NETWORK
TITLE = Hys Calculation
//Level Hys Absolute
      L     #Param.L_Hi_Lim;
      L     #Param.L_Lo_Lim;
      -R;
      L     100.0;
      /R;
      L     #Param.L_Hys;
      *R;
      T     #L_Hys_Abs;
//Tank High Level
      L     #Param.SP_Level_HL;
      L     #L_Hys_Abs;
      -R;
      T     #Hys_Level_HL;
//Tank Mid Level
      L     #Param.SP_Level_ML;
      L     #L_Hys_Abs;
      -R;
      T     #Hys_Level_ML;
//Tank Low Level
      L     #Param.SP_Level_LL;
      L     #L_Hys_Abs;
      +R;
      T     #Hys_Level_LL;


REGION Network 3: Level Tank
   RUNG wire#powerrail
      Contact( #alwaysON )
      wire#w1
      { S7_Templates := "SrcType := Real" } LE_Contact(in1 := #Param.SP_Level_HL, in2 := #IN_LT01)
      S_Coil( #State.Tank_HL )
   END_RUNG
   RUNG wire#w1
      { S7_Templates := "SrcType := Real" } GT_Contact(in1 := #Hys_Level_HL, in2 := #IN_LT01)
      R_Coil( #State.Tank_HL )
   END_RUNG
   RUNG wire#w1
      { S7_Templates := "SrcType := Real" } LE_Contact(in1 := #Param.SP_Level_ML, in2 := #IN_LT01)
      S_Coil( #State.Tank_ML )
   END_RUNG
   RUNG wire#w1
      { S7_Templates := "SrcType := Real" } GT_Contact(in1 := #Hys_Level_ML, in2 := #IN_LT01)
      R_Coil( #State.Tank_ML )
   END_RUNG
   RUNG wire#w1
      { S7_Templates := "SrcType := Real" } GE_Contact(in1 := #Param.SP_Level_LL, in2 := #IN_LT01)
      S_Coil( #State.Tank_LL )
   END_RUNG
   RUNG wire#w1
      { S7_Templates := "SrcType := Real" } LT_Contact(in1 := #Hys_Level_LL, in2 := #IN_LT01)
      R_Coil( #State.Tank_LL )
   END_RUNG
   // the same network as SCL:
   IF #alwaysON AND (#Param.SP_Level_HL <= #IN_LT01) THEN #State.Tank_HL := TRUE; END_IF;
   IF #alwaysON AND (#Hys_Level_HL > #IN_LT01) THEN #State.Tank_HL := FALSE; END_IF;
   IF #alwaysON AND (#Param.SP_Level_ML <= #IN_LT01) THEN #State.Tank_ML := TRUE; END_IF;
   IF #alwaysON AND (#Hys_Level_ML > #IN_LT01) THEN #State.Tank_ML := FALSE; END_IF;
   IF #alwaysON AND (#Param.SP_Level_LL >= #IN_LT01) THEN #State.Tank_LL := TRUE; END_IF;
   IF #alwaysON AND (#Hys_Level_LL < #IN_LT01) THEN #State.Tank_LL := FALSE; END_IF;
END_REGION

REGION Network 4: Reset Command Inload
   RUNG wire#powerrail
      Contact( #alwaysON )
      Contact( #State.Tank_HL )
      P_Trig( #r.PosE1 )
      wire#w1
      R_Coil( #Cmd.Inload )
   END_RUNG
   RUNG wire#w1
      R_Coil( #Actuator.LCS_OnOff )
   END_RUNG
   // the same network as SCL:
   #_w1 := #alwaysON AND #State.Tank_HL;
   #_w2 := #_w1 AND NOT #r.PosE1;   // rising edge
   #r.PosE1 := #_w1;
   IF #_w2 THEN
       #Cmd.Inload := FALSE;
       #Actuator.LCS_OnOff := FALSE;
   END_IF;
END_REGION

REGION Network 5: Inload from LCS ON-OFF
   RUNG wire#powerrail
      Contact( #alwaysON )
      wire#w1
      Contact( #"LCS Start" )
      S_Coil( #Actuator.LCS_OnOff )
   END_RUNG
   RUNG wire#w1
      Contact( #"LCS Stop" )
      R_Coil( #Actuator.LCS_OnOff )
   END_RUNG
   // the same network as SCL:
   IF #alwaysON AND #"LCS Start" THEN #Actuator.LCS_OnOff := TRUE; END_IF;
   IF #alwaysON AND #"LCS Stop" THEN #Actuator.LCS_OnOff := FALSE; END_IF;
END_REGION

REGION Network 6: Command Inload Material to Buffer Tank
   RUNG wire#powerrail
      Contact( #alwaysON )
      wire#w1
      I_Contact( #State.Tank_HL )
      I_Contact( #"Inload Busy" )
      I_Contact( #State.Tank_inCIP )
      I_Contact( #State.Line_inCIP )
      Coil( #State.Inload_Enable )
   END_RUNG
   RUNG wire#w1
      Contact( #State.Inload_Enable )
      wire#w2
      Contact( #Cmd.Inload )
      wire#w3
      S_Coil( #State.Inloading )
   END_RUNG
   RUNG wire#w2
      Contact( #Actuator.LCS_OnOff )
   END_RUNG wire#w3
   RUNG wire#w1
      I_Contact( #State.Inload_Enable )
      R_Coil( #Cmd.Inload )
   END_RUNG
   RUNG wire#w1
      I_Contact( #Cmd.Inload )
      I_Contact( #Actuator.LCS_OnOff )
      R_Coil( #State.Inloading )
   END_RUNG
   // the same network as SCL:
   #State.Inload_Enable := #alwaysON AND NOT #State.Tank_HL AND NOT #"Inload Busy" AND NOT #State.Tank_inCIP AND NOT #State.Line_inCIP;
   IF #alwaysON AND #State.Inload_Enable AND (#Cmd.Inload OR #Actuator.LCS_OnOff) THEN
       #State.Inloading := TRUE;
   END_IF;
   IF #alwaysON AND NOT #State.Inload_Enable THEN #Cmd.Inload := FALSE; END_IF;
   IF #alwaysON AND NOT #Cmd.Inload AND NOT #Actuator.LCS_OnOff THEN #State.Inloading := FALSE; END_IF;
END_REGION

REGION Network 7: Tank Ready for Transfer to Blending
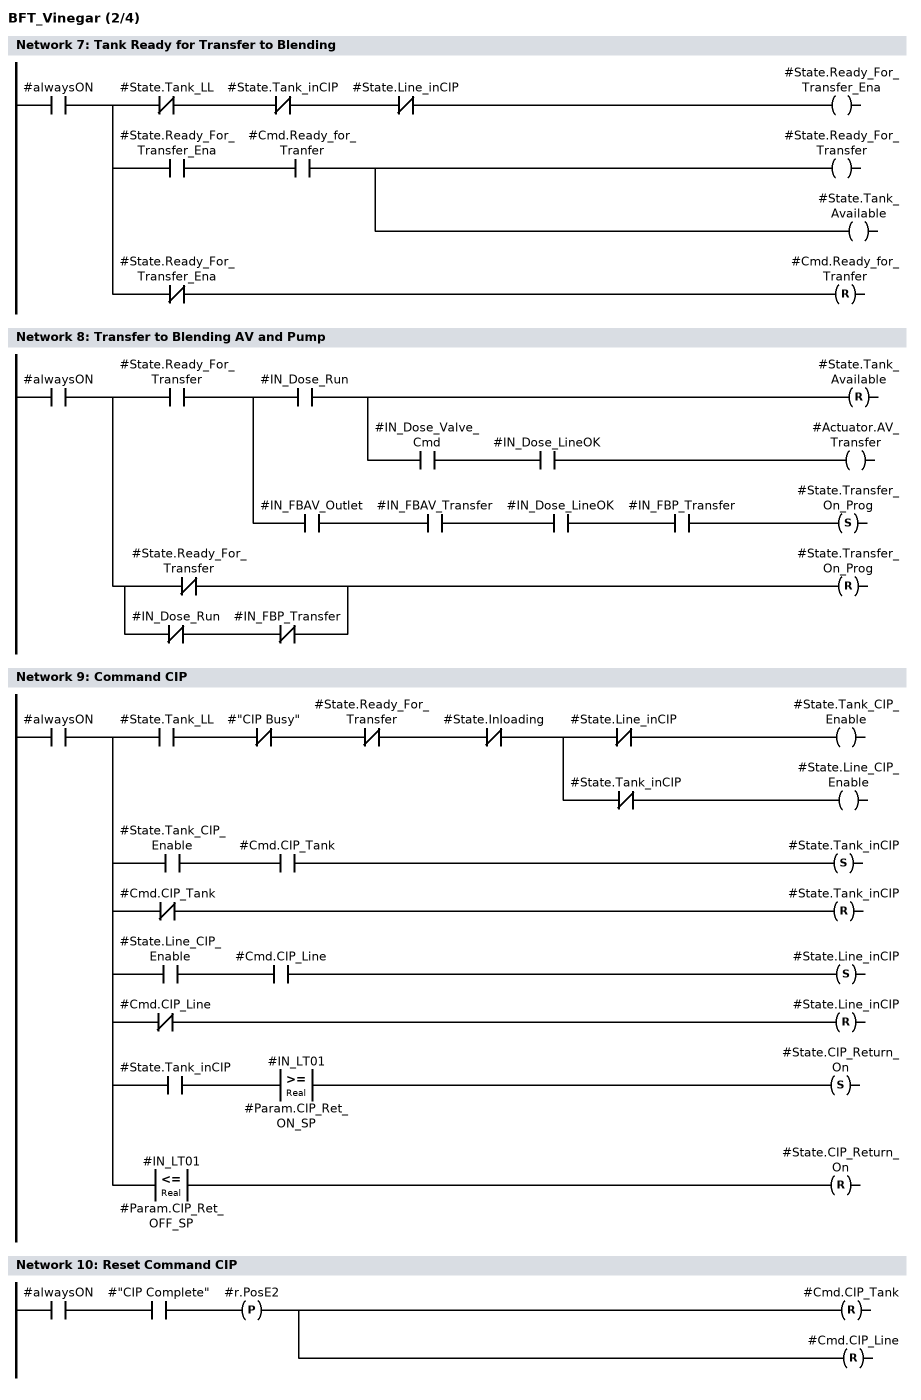
   RUNG wire#powerrail
      Contact( #alwaysON )
      wire#w1
      I_Contact( #State.Tank_LL )
      I_Contact( #State.Tank_inCIP )
      I_Contact( #State.Line_inCIP )
      Coil( #State.Ready_For_Transfer_Ena )
   END_RUNG
   RUNG wire#w1
      Contact( #State.Ready_For_Transfer_Ena )
      Contact( #Cmd.Ready_for_Tranfer )
      wire#w2
      Coil( #State.Ready_For_Transfer )
   END_RUNG
   RUNG wire#w2
      Coil( #State.Tank_Available )
   END_RUNG
   RUNG wire#w1
      I_Contact( #State.Ready_For_Transfer_Ena )
      R_Coil( #Cmd.Ready_for_Tranfer )
   END_RUNG
   // the same network as SCL:
   #State.Ready_For_Transfer_Ena := #alwaysON AND NOT #State.Tank_LL AND NOT #State.Tank_inCIP AND NOT #State.Line_inCIP;
   #State.Ready_For_Transfer := #alwaysON AND #State.Ready_For_Transfer_Ena AND #Cmd.Ready_for_Tranfer;
   #State.Tank_Available := #State.Ready_For_Transfer;
   IF #alwaysON AND NOT #State.Ready_For_Transfer_Ena THEN #Cmd.Ready_for_Tranfer := FALSE; END_IF;
END_REGION

REGION Network 8: Transfer to Blending AV and Pump
   RUNG wire#powerrail
      Contact( #alwaysON )
      wire#w1
      Contact( #State.Ready_For_Transfer )
      wire#w2
      Contact( #IN_Dose_Run )
      wire#w3
      R_Coil( #State.Tank_Available )
   END_RUNG
   RUNG wire#w3
      Contact( #IN_Dose_Valve_Cmd )
      Contact( #IN_Dose_LineOK )
      Coil( #Actuator.AV_Transfer )
   END_RUNG
   RUNG wire#w2
      Contact( #IN_FBAV_Outlet )
      Contact( #IN_FBAV_Transfer )
      Contact( #IN_Dose_LineOK )
      Contact( #IN_FBP_Transfer )
      S_Coil( #State.Transfer_On_Prog )
   END_RUNG
   RUNG wire#w1
      I_Contact( #State.Ready_For_Transfer )
      wire#w4
      R_Coil( #State.Transfer_On_Prog )
   END_RUNG
   RUNG wire#w1
      I_Contact( #IN_Dose_Run )
      I_Contact( #IN_FBP_Transfer )
   END_RUNG wire#w4
   // the same network as SCL:
   #_w1 := #alwaysON AND #State.Ready_For_Transfer;
   #_w2 := #_w1 AND #IN_Dose_Run;
   IF #_w2 THEN #State.Tank_Available := FALSE; END_IF;
   #Actuator.AV_Transfer := #_w2 AND #IN_Dose_Valve_Cmd AND #IN_Dose_LineOK;
   IF #_w1 AND #IN_FBAV_Outlet AND #IN_FBAV_Transfer AND #IN_Dose_LineOK AND #IN_FBP_Transfer THEN
       #State.Transfer_On_Prog := TRUE;
   END_IF;
   IF #alwaysON AND (NOT #State.Ready_For_Transfer OR (NOT #IN_Dose_Run AND NOT #IN_FBP_Transfer)) THEN
       #State.Transfer_On_Prog := FALSE;
   END_IF;
END_REGION

REGION Network 9: Command CIP
   RUNG wire#powerrail
      Contact( #alwaysON )
      wire#w1
      Contact( #State.Tank_LL )
      I_Contact( #"CIP Busy" )
      I_Contact( #State.Ready_For_Transfer )
      I_Contact( #State.Inloading )
      wire#w2
      I_Contact( #State.Line_inCIP )
      Coil( #State.Tank_CIP_Enable )
   END_RUNG
   RUNG wire#w2
      I_Contact( #State.Tank_inCIP )
      Coil( #State.Line_CIP_Enable )
   END_RUNG
   RUNG wire#w1
      Contact( #State.Tank_CIP_Enable )
      Contact( #Cmd.CIP_Tank )
      S_Coil( #State.Tank_inCIP )
   END_RUNG
   RUNG wire#w1
      I_Contact( #Cmd.CIP_Tank )
      R_Coil( #State.Tank_inCIP )
   END_RUNG
   RUNG wire#w1
      Contact( #State.Line_CIP_Enable )
      Contact( #Cmd.CIP_Line )
      S_Coil( #State.Line_inCIP )
   END_RUNG
   RUNG wire#w1
      I_Contact( #Cmd.CIP_Line )
      R_Coil( #State.Line_inCIP )
   END_RUNG
   RUNG wire#w1
      Contact( #State.Tank_inCIP )
      { S7_Templates := "SrcType := Real" } GE_Contact(in1 := #IN_LT01, in2 := #Param.CIP_Ret_ON_SP)
      S_Coil( #State.CIP_Return_On )
   END_RUNG
   RUNG wire#w1
      { S7_Templates := "SrcType := Real" } LE_Contact(in1 := #IN_LT01, in2 := #Param.CIP_Ret_OFF_SP)
      R_Coil( #State.CIP_Return_On )
   END_RUNG
   // the same network as SCL:
   #_w1 := #alwaysON AND #State.Tank_LL AND NOT #"CIP Busy" AND NOT #State.Ready_For_Transfer AND NOT #State.Inloading;
   #State.Tank_CIP_Enable := #_w1 AND NOT #State.Line_inCIP;
   #State.Line_CIP_Enable := #_w1 AND NOT #State.Tank_inCIP;
   IF #alwaysON AND #State.Tank_CIP_Enable AND #Cmd.CIP_Tank THEN #State.Tank_inCIP := TRUE; END_IF;
   IF #alwaysON AND NOT #Cmd.CIP_Tank THEN #State.Tank_inCIP := FALSE; END_IF;
   IF #alwaysON AND #State.Line_CIP_Enable AND #Cmd.CIP_Line THEN #State.Line_inCIP := TRUE; END_IF;
   IF #alwaysON AND NOT #Cmd.CIP_Line THEN #State.Line_inCIP := FALSE; END_IF;
   IF #alwaysON AND #State.Tank_inCIP AND (#IN_LT01 >= #Param.CIP_Ret_ON_SP) THEN
       #State.CIP_Return_On := TRUE;
   END_IF;
   IF #alwaysON AND (#IN_LT01 <= #Param.CIP_Ret_OFF_SP) THEN #State.CIP_Return_On := FALSE; END_IF;
END_REGION

REGION Network 10: Reset Command CIP
   RUNG wire#powerrail
      Contact( #alwaysON )
      Contact( #"CIP Complete" )
      P_Trig( #r.PosE2 )
      wire#w1
      R_Coil( #Cmd.CIP_Tank )
   END_RUNG
   RUNG wire#w1
      R_Coil( #Cmd.CIP_Line )
   END_RUNG
   // the same network as SCL:
   #_w1 := #alwaysON AND #"CIP Complete";
   #_w2 := #_w1 AND NOT #r.PosE2;   // rising edge
   #r.PosE2 := #_w1;
   IF #_w2 THEN
       #Cmd.CIP_Tank := FALSE;
       #Cmd.CIP_Line := FALSE;
   END_IF;
END_REGION

REGION Network 11: CIP Request and CIP Line Open
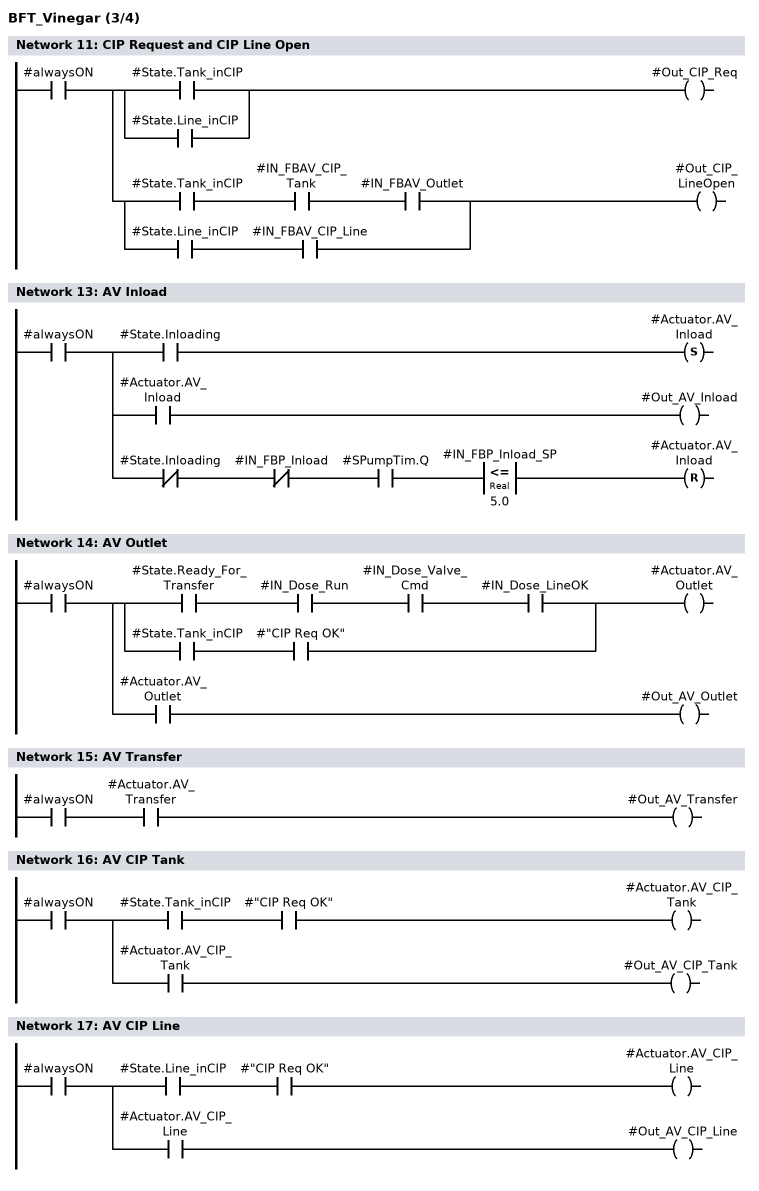
   RUNG wire#powerrail
      Contact( #alwaysON )
      wire#w1
      Contact( #State.Tank_inCIP )
      wire#w2
      Coil( #Out_CIP_Req )
   END_RUNG
   RUNG wire#w1
      Contact( #State.Line_inCIP )
   END_RUNG wire#w2
   RUNG wire#w1
      Contact( #State.Tank_inCIP )
      Contact( #IN_FBAV_CIP_Tank )
      Contact( #IN_FBAV_Outlet )
      wire#w3
      Coil( #Out_CIP_LineOpen )
   END_RUNG
   RUNG wire#w1
      Contact( #State.Line_inCIP )
      Contact( #IN_FBAV_CIP_Line )
   END_RUNG wire#w3
   // the same network as SCL:
   #Out_CIP_Req := #alwaysON AND (#State.Tank_inCIP OR #State.Line_inCIP);
   #Out_CIP_LineOpen := #alwaysON AND ((#State.Tank_inCIP AND #IN_FBAV_CIP_Tank AND #IN_FBAV_Outlet) OR (#State.Line_inCIP AND #IN_FBAV_CIP_Line));
END_REGION

REGION Network 13: AV Inload
   RUNG wire#powerrail
      Contact( #alwaysON )
      wire#w1
      Contact( #State.Inloading )
      S_Coil( #Actuator.AV_Inload )
   END_RUNG
   RUNG wire#w1
      Contact( #Actuator.AV_Inload )
      Coil( #Out_AV_Inload )
   END_RUNG
   RUNG wire#w1
      I_Contact( #State.Inloading )
      I_Contact( #IN_FBP_Inload )
      Contact( #SPumpTim.Q )
      { S7_Templates := "SrcType := Real" } LE_Contact(in1 := #IN_FBP_Inload_SP, in2 := 5.0)
      R_Coil( #Actuator.AV_Inload )
   END_RUNG
   // the same network as SCL:
   IF #alwaysON AND #State.Inloading THEN #Actuator.AV_Inload := TRUE; END_IF;
   #Out_AV_Inload := #alwaysON AND #Actuator.AV_Inload;
   IF #alwaysON AND NOT #State.Inloading AND NOT #IN_FBP_Inload AND #SPumpTim.Q AND (#IN_FBP_Inload_SP <= 5.0) THEN
       #Actuator.AV_Inload := FALSE;
   END_IF;
END_REGION

REGION Network 14: AV Outlet
   RUNG wire#powerrail
      Contact( #alwaysON )
      wire#w1
      Contact( #State.Ready_For_Transfer )
      Contact( #IN_Dose_Run )
      Contact( #IN_Dose_Valve_Cmd )
      Contact( #IN_Dose_LineOK )
      wire#w2
      Coil( #Actuator.AV_Outlet )
   END_RUNG
   RUNG wire#w1
      Contact( #State.Tank_inCIP )
      Contact( #"CIP Req OK" )
   END_RUNG wire#w2
   RUNG wire#w1
      Contact( #Actuator.AV_Outlet )
      Coil( #Out_AV_Outlet )
   END_RUNG
   // the same network as SCL:
   #Actuator.AV_Outlet := #alwaysON AND ((#State.Ready_For_Transfer AND #IN_Dose_Run AND #IN_Dose_Valve_Cmd AND #IN_Dose_LineOK) OR (#State.Tank_inCIP AND #"CIP Req OK"));
   #Out_AV_Outlet := #alwaysON AND #Actuator.AV_Outlet;
END_REGION

REGION Network 15: AV Transfer
   RUNG wire#powerrail
      Contact( #alwaysON )
      Contact( #Actuator.AV_Transfer )
      Coil( #Out_AV_Transfer )
   END_RUNG
   // the same network as SCL:
   #Out_AV_Transfer := #alwaysON AND #Actuator.AV_Transfer;
END_REGION

REGION Network 16: AV CIP Tank
   RUNG wire#powerrail
      Contact( #alwaysON )
      wire#w1
      Contact( #State.Tank_inCIP )
      Contact( #"CIP Req OK" )
      Coil( #Actuator.AV_CIP_Tank )
   END_RUNG
   RUNG wire#w1
      Contact( #Actuator.AV_CIP_Tank )
      Coil( #Out_AV_CIP_Tank )
   END_RUNG
   // the same network as SCL:
   #Actuator.AV_CIP_Tank := #alwaysON AND #State.Tank_inCIP AND #"CIP Req OK";
   #Out_AV_CIP_Tank := #alwaysON AND #Actuator.AV_CIP_Tank;
END_REGION

REGION Network 17: AV CIP Line
   RUNG wire#powerrail
      Contact( #alwaysON )
      wire#w1
      Contact( #State.Line_inCIP )
      Contact( #"CIP Req OK" )
      Coil( #Actuator.AV_CIP_Line )
   END_RUNG
   RUNG wire#w1
      Contact( #Actuator.AV_CIP_Line )
      Coil( #Out_AV_CIP_Line )
   END_RUNG
   // the same network as SCL:
   #Actuator.AV_CIP_Line := #alwaysON AND #State.Line_inCIP AND #"CIP Req OK";
   #Out_AV_CIP_Line := #alwaysON AND #Actuator.AV_CIP_Line;
END_REGION

REGION Network 19: Pump Inload
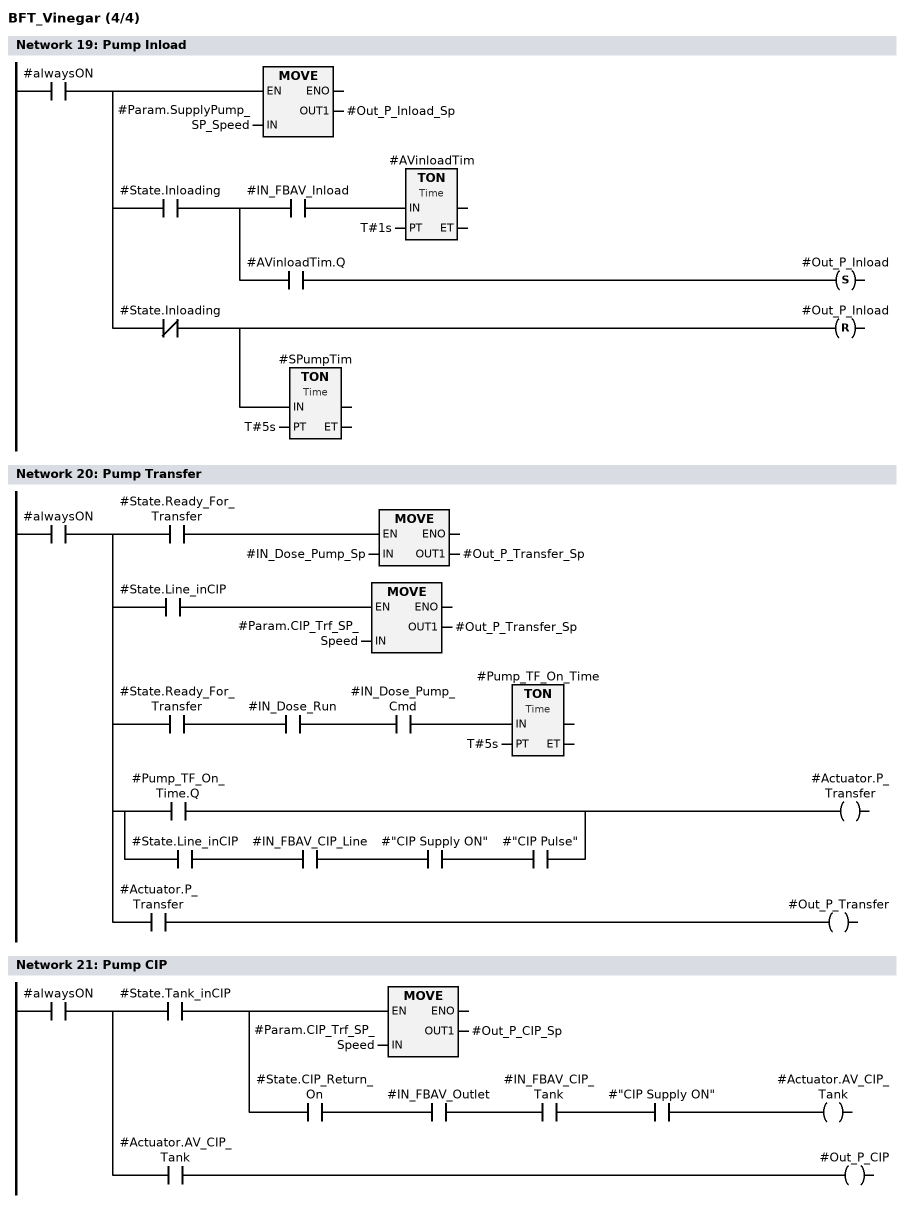
   RUNG wire#powerrail
      Contact( #alwaysON )
      wire#w1
      Move(in := #Param.SupplyPump_SP_Speed, out1 => #Out_P_Inload_Sp)
   END_RUNG
   RUNG wire#w1
      Contact( #State.Inloading )
      wire#w2
      Contact( #IN_FBAV_Inload )
      { S7_Templates := "time_type := Time" } #AVinloadTim.TON(pt := T#1s, et =>)
   END_RUNG
   RUNG wire#w2
      Contact( #AVinloadTim.Q )
      S_Coil( #Out_P_Inload )
   END_RUNG
   RUNG wire#w1
      I_Contact( #State.Inloading )
      wire#w3
      R_Coil( #Out_P_Inload )
   END_RUNG
   RUNG wire#w3
      { S7_Templates := "time_type := Time" } #SPumpTim.TON(pt := T#5s, et =>)
   END_RUNG
   // the same network as SCL:
   IF #alwaysON THEN #Out_P_Inload_Sp := #Param.SupplyPump_SP_Speed; END_IF;
   #_w1 := #alwaysON AND #State.Inloading;
   #AVinloadTim(IN := #_w1 AND #IN_FBAV_Inload, PT := T#1s);   // TON
   IF #_w1 AND #AVinloadTim.Q THEN #Out_P_Inload := TRUE; END_IF;
   #_w2 := #alwaysON AND NOT #State.Inloading;
   IF #_w2 THEN #Out_P_Inload := FALSE; END_IF;
   #SPumpTim(IN := #_w2, PT := T#5s);   // TON
END_REGION

REGION Network 20: Pump Transfer
   RUNG wire#powerrail
      Contact( #alwaysON )
      wire#w1
      Contact( #State.Ready_For_Transfer )
      Move(in := #IN_Dose_Pump_Sp, out1 => #Out_P_Transfer_Sp)
   END_RUNG
   RUNG wire#w1
      Contact( #State.Line_inCIP )
      Move(in := #Param.CIP_Trf_SP_Speed, out1 => #Out_P_Transfer_Sp)
   END_RUNG
   RUNG wire#w1
      Contact( #State.Ready_For_Transfer )
      Contact( #IN_Dose_Run )
      Contact( #IN_Dose_Pump_Cmd )
      { S7_Templates := "time_type := Time" } #Pump_TF_On_Time.TON(pt := T#5s, et =>)
   END_RUNG
   RUNG wire#w1
      Contact( #Pump_TF_On_Time.Q )
      wire#w2
      Coil( #Actuator.P_Transfer )
   END_RUNG
   RUNG wire#w1
      Contact( #State.Line_inCIP )
      Contact( #IN_FBAV_CIP_Line )
      Contact( #"CIP Supply ON" )
      Contact( #"CIP Pulse" )
   END_RUNG wire#w2
   RUNG wire#w1
      Contact( #Actuator.P_Transfer )
      Coil( #Out_P_Transfer )
   END_RUNG
   // the same network as SCL:
   IF #alwaysON AND #State.Ready_For_Transfer THEN #Out_P_Transfer_Sp := #IN_Dose_Pump_Sp; END_IF;
   IF #alwaysON AND #State.Line_inCIP THEN #Out_P_Transfer_Sp := #Param.CIP_Trf_SP_Speed; END_IF;
   #Pump_TF_On_Time(IN := #alwaysON AND #State.Ready_For_Transfer AND #IN_Dose_Run AND #IN_Dose_Pump_Cmd,   // TON
                    PT := T#5s);
   #Actuator.P_Transfer := #alwaysON AND (#Pump_TF_On_Time.Q OR (#State.Line_inCIP AND #IN_FBAV_CIP_Line AND #"CIP Supply ON" AND #"CIP Pulse"));
   #Out_P_Transfer := #alwaysON AND #Actuator.P_Transfer;
END_REGION

REGION Network 21: Pump CIP
   RUNG wire#powerrail
      Contact( #alwaysON )
      wire#w1
      Contact( #State.Tank_inCIP )
      wire#w2
      Move(in := #Param.CIP_Trf_SP_Speed, out1 => #Out_P_CIP_Sp)
   END_RUNG
   RUNG wire#w2
      Contact( #State.CIP_Return_On )
      Contact( #IN_FBAV_Outlet )
      Contact( #IN_FBAV_CIP_Tank )
      Contact( #"CIP Supply ON" )
      Coil( #Actuator.AV_CIP_Tank )
   END_RUNG
   RUNG wire#w1
      Contact( #Actuator.AV_CIP_Tank )
      Coil( #Out_P_CIP )
   END_RUNG
   // the same network as SCL:
   #_w1 := #alwaysON AND #State.Tank_inCIP;
   IF #_w1 THEN #Out_P_CIP_Sp := #Param.CIP_Trf_SP_Speed; END_IF;
   #Actuator.AV_CIP_Tank := #_w1 AND #State.CIP_Return_On AND #IN_FBAV_Outlet AND #IN_FBAV_CIP_Tank AND #"CIP Supply ON";
   #Out_P_CIP := #alwaysON AND #Actuator.AV_CIP_Tank;
END_REGION
END_FUNCTION_BLOCK

FUNCTION_BLOCK "Hot_Water"   // FB366, LAD
{ S7_Optimized_Access := 'TRUE' }
VERSION : 0.1
// stored: AutoNumber false, IsIECCheckEnabled false, IsRetainMemResEnabled false, MemoryReserve 100, SetENOAutomatically false, UDAEnableTagReadback false
   VAR_INPUT
      IN_FBAV_Inload : Bool;
      IN_FBAV_Outlet : Bool;
      IN_FBAV_Transfer : Bool;
      IN_FBP_Transfer : Bool;
      IN_FBP_Transfer_SP : Real;
      IN_Dose_Run : Bool;
      IN_Dose_Held : Bool;
      IN_Dose_Complete : Bool;
      IN_Dose_Header_1 : Bool;
      IN_Dose_Header_2 : Bool;
      IN_Dose_Valve_Cmd : Bool;
      IN_Dose_Pump_Cmd : Bool;
      IN_Dose_Pump_Sp : Real;
      IN_Dose_LineOK : Bool;
      IN_Low_Level : Bool;
      IN_Med_Level : Bool;
      IN_High_Level : Bool;
      IN_FBCV : Bool;
      "IN_FBCV_Act%" : Real;
      IN_Temperature : Real;
   END_VAR
   VAR_OUTPUT
      Out_AV_Inload : Bool;
      Out_AV_Outlet : Bool;
      Out_AV_Transfer : Bool;
      Out_P_Transfer : Bool;
      Out_P_Transfer_Sp : Real;
      OUT_CV : Bool;
      Out_Temp_Act : Real;
      Out_Temp_Sp : Real;
   END_VAR
   VAR
      Cmd : Struct
         Inload_Start : Bool;
         Inload_Mode : Bool := 1;   // 0 : Manual ;; 1 : Auto
         ReadyForTransfer : Bool;
         Transfer_Mode : Bool;   // 0 : By Timer ;; 1 : By Quantity
      END_STRUCT;
   END_VAR
   VAR RETAIN
      Param : Struct
         Temperature_SP : Real := 50.0;
      END_STRUCT;
   END_VAR
   VAR
      State : Struct
         Tank_LL : Bool;
         Tank_ML : Bool;
         Tank_HL : Bool;
         Inload_EN : Bool;
         Inload_Aut : Bool;
         Inloading : Bool;
         Ready_For_Transfer_EN : Bool;
         Ready_For_Transfer : Bool;
         Tank_Available : Bool;
         Transfer_on_Prog : Bool;
      END_STRUCT;
      alwaysON : Bool;
      r : Struct
         PosE1 : Bool;
         PosE2 : Bool;
         PosE3 : Bool;
         PosE4 : Bool;
         PosE5 : Bool;
         PosE6 : Bool;
         PosE7 : Bool;
         PosE8 : Bool;
         PosE9 : Bool;
         PosE10 : Bool;
         PosE11 : Bool;
         PosE12 : Bool;
         PosE13 : Bool;
         PosE14 : Bool;
         PosE15 : Bool;
         PosE16 : Bool;
         PosE17 : Bool;
         PosE18 : Bool;
         PosE19 : Bool;
         PosE20 : Bool;
         PosE21 : Bool;
         PosE22 : Bool;
         PosE23 : Bool;
         PosE24 : Bool;
         PosE25 : Bool;
         PosE26 : Bool;
         PosE27 : Bool;
         PosE28 : Bool;
         PosE29 : Bool;
         PosE30 : Bool;
         PosE31 : Bool;
         PosE32 : Bool;
      END_STRUCT;
      Actuator : Struct
         AV_Inload : Bool;
         AV_Outlet : Bool;
         AV_Transfer : Bool;
         AV_CIP_Tank : Bool;
         AV_CIP_Line : Bool;
         P_Transfer : Bool;
         P_Inload : Bool;
         P_CIP : Bool;
         CV : Bool;
      END_STRUCT;
      SPumpTim { S7_SetPoint := 'True'} : TON_TIME;
   END_VAR
   VAR_TEMP   // added for the SCL form of the ladder/FBD networks
      _w1 : Bool;
      _w2 : Bool;
   END_VAR
BEGIN

REGION Network 1: Always_ON
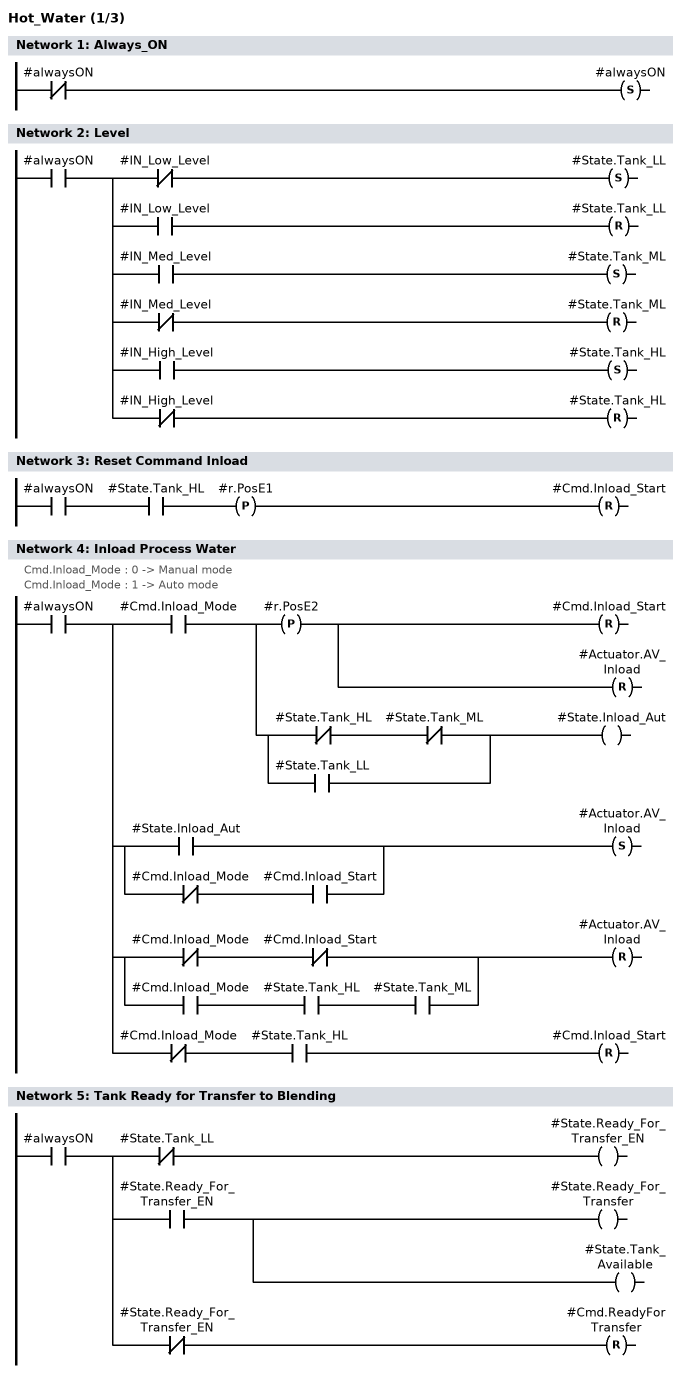
   RUNG wire#powerrail
      I_Contact( #alwaysON )
      S_Coil( #alwaysON )
   END_RUNG
   // the same network as SCL:
   IF NOT #alwaysON THEN #alwaysON := TRUE; END_IF;
END_REGION

REGION Network 2: Level
   RUNG wire#powerrail
      Contact( #alwaysON )
      wire#w1
      I_Contact( #IN_Low_Level )
      S_Coil( #State.Tank_LL )
   END_RUNG
   RUNG wire#w1
      Contact( #IN_Low_Level )
      R_Coil( #State.Tank_LL )
   END_RUNG
   RUNG wire#w1
      Contact( #IN_Med_Level )
      S_Coil( #State.Tank_ML )
   END_RUNG
   RUNG wire#w1
      I_Contact( #IN_Med_Level )
      R_Coil( #State.Tank_ML )
   END_RUNG
   RUNG wire#w1
      Contact( #IN_High_Level )
      S_Coil( #State.Tank_HL )
   END_RUNG
   RUNG wire#w1
      I_Contact( #IN_High_Level )
      R_Coil( #State.Tank_HL )
   END_RUNG
   // the same network as SCL:
   IF #alwaysON AND NOT #IN_Low_Level THEN #State.Tank_LL := TRUE; END_IF;
   IF #alwaysON AND #IN_Low_Level THEN #State.Tank_LL := FALSE; END_IF;
   IF #alwaysON AND #IN_Med_Level THEN #State.Tank_ML := TRUE; END_IF;
   IF #alwaysON AND NOT #IN_Med_Level THEN #State.Tank_ML := FALSE; END_IF;
   IF #alwaysON AND #IN_High_Level THEN #State.Tank_HL := TRUE; END_IF;
   IF #alwaysON AND NOT #IN_High_Level THEN #State.Tank_HL := FALSE; END_IF;
END_REGION

REGION Network 3: Reset Command Inload
   RUNG wire#powerrail
      Contact( #alwaysON )
      Contact( #State.Tank_HL )
      P_Trig( #r.PosE1 )
      R_Coil( #Cmd.Inload_Start )
   END_RUNG
   // the same network as SCL:
   #_w1 := #alwaysON AND #State.Tank_HL;
   #_w2 := #_w1 AND NOT #r.PosE1;   // rising edge
   #r.PosE1 := #_w1;
   IF #_w2 THEN #Cmd.Inload_Start := FALSE; END_IF;
END_REGION

REGION Network 4: Inload Process Water
   // Cmd.Inload_Mode : 0 -> Manual mode
   // Cmd.Inload_Mode : 1 -> Auto mode
   RUNG wire#powerrail
      Contact( #alwaysON )
      wire#w1
      Contact( #Cmd.Inload_Mode )
      wire#w2
      P_Trig( #r.PosE2 )
      wire#w3
      R_Coil( #Cmd.Inload_Start )
   END_RUNG
   RUNG wire#w3
      R_Coil( #Actuator.AV_Inload )
   END_RUNG
   RUNG wire#w2
      I_Contact( #State.Tank_HL )
      I_Contact( #State.Tank_ML )
      wire#w4
      Coil( #State.Inload_Aut )
   END_RUNG
   RUNG wire#w2
      Contact( #State.Tank_LL )
   END_RUNG wire#w4
   RUNG wire#w1
      Contact( #State.Inload_Aut )
      wire#w5
      S_Coil( #Actuator.AV_Inload )
   END_RUNG
   RUNG wire#w1
      I_Contact( #Cmd.Inload_Mode )
      Contact( #Cmd.Inload_Start )
   END_RUNG wire#w5
   RUNG wire#w1
      I_Contact( #Cmd.Inload_Mode )
      I_Contact( #Cmd.Inload_Start )
      wire#w6
      R_Coil( #Actuator.AV_Inload )
   END_RUNG
   RUNG wire#w1
      Contact( #Cmd.Inload_Mode )
      Contact( #State.Tank_HL )
      Contact( #State.Tank_ML )
   END_RUNG wire#w6
   RUNG wire#w1
      I_Contact( #Cmd.Inload_Mode )
      Contact( #State.Tank_HL )
      R_Coil( #Cmd.Inload_Start )
   END_RUNG
   // the same network as SCL:
   #_w1 := #alwaysON AND #Cmd.Inload_Mode;
   #_w2 := #_w1 AND NOT #r.PosE2;   // rising edge
   #r.PosE2 := #_w1;
   IF #_w2 THEN
       #Cmd.Inload_Start := FALSE;
       #Actuator.AV_Inload := FALSE;
   END_IF;
   #State.Inload_Aut := #_w1 AND ((NOT #State.Tank_HL AND NOT #State.Tank_ML) OR #State.Tank_LL);
   IF #alwaysON AND (#State.Inload_Aut OR (NOT #Cmd.Inload_Mode AND #Cmd.Inload_Start)) THEN
       #Actuator.AV_Inload := TRUE;
   END_IF;
   IF #alwaysON AND ((NOT #Cmd.Inload_Mode AND NOT #Cmd.Inload_Start) OR (#Cmd.Inload_Mode AND #State.Tank_HL AND #State.Tank_ML)) THEN
       #Actuator.AV_Inload := FALSE;
   END_IF;
   IF #alwaysON AND NOT #Cmd.Inload_Mode AND #State.Tank_HL THEN #Cmd.Inload_Start := FALSE; END_IF;
END_REGION

REGION Network 5: Tank Ready for Transfer to Blending
   RUNG wire#powerrail
      Contact( #alwaysON )
      wire#w1
      I_Contact( #State.Tank_LL )
      Coil( #State.Ready_For_Transfer_EN )
   END_RUNG
   RUNG wire#w1
      Contact( #State.Ready_For_Transfer_EN )
      wire#w2
      Coil( #State.Ready_For_Transfer )
   END_RUNG
   RUNG wire#w2
      Coil( #State.Tank_Available )
   END_RUNG
   RUNG wire#w1
      I_Contact( #State.Ready_For_Transfer_EN )
      R_Coil( #Cmd.ReadyForTransfer )
   END_RUNG
   // the same network as SCL:
   #State.Ready_For_Transfer_EN := #alwaysON AND NOT #State.Tank_LL;
   #State.Ready_For_Transfer := #alwaysON AND #State.Ready_For_Transfer_EN;
   #State.Tank_Available := #State.Ready_For_Transfer;
   IF #alwaysON AND NOT #State.Ready_For_Transfer_EN THEN #Cmd.ReadyForTransfer := FALSE; END_IF;
END_REGION

REGION Network 6: Transfer to Blending AV and Pump
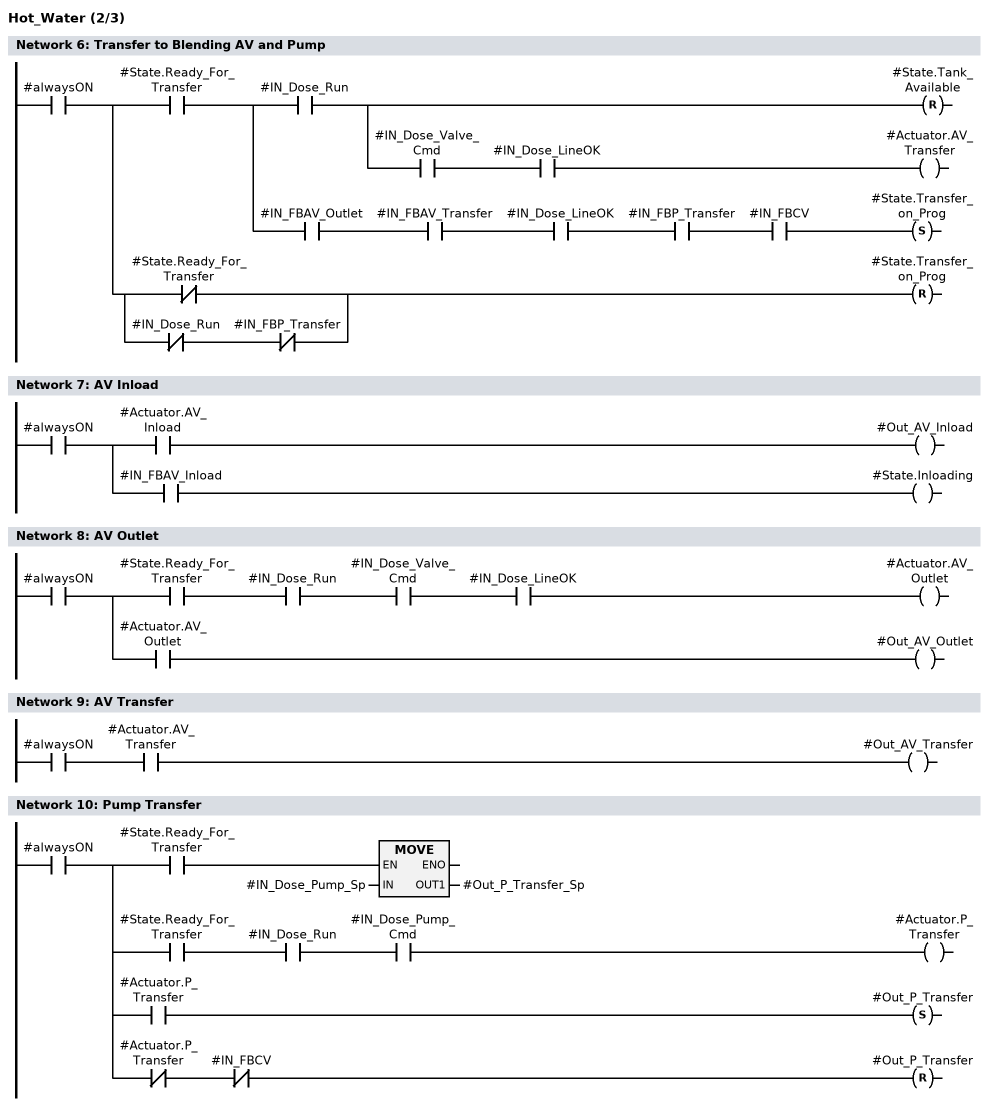
   RUNG wire#powerrail
      Contact( #alwaysON )
      wire#w1
      Contact( #State.Ready_For_Transfer )
      wire#w2
      Contact( #IN_Dose_Run )
      wire#w3
      R_Coil( #State.Tank_Available )
   END_RUNG
   RUNG wire#w3
      Contact( #IN_Dose_Valve_Cmd )
      Contact( #IN_Dose_LineOK )
      Coil( #Actuator.AV_Transfer )
   END_RUNG
   RUNG wire#w2
      Contact( #IN_FBAV_Outlet )
      Contact( #IN_FBAV_Transfer )
      Contact( #IN_Dose_LineOK )
      Contact( #IN_FBP_Transfer )
      Contact( #IN_FBCV )
      S_Coil( #State.Transfer_on_Prog )
   END_RUNG
   RUNG wire#w1
      I_Contact( #State.Ready_For_Transfer )
      wire#w4
      R_Coil( #State.Transfer_on_Prog )
   END_RUNG
   RUNG wire#w1
      I_Contact( #IN_Dose_Run )
      I_Contact( #IN_FBP_Transfer )
   END_RUNG wire#w4
   // the same network as SCL:
   #_w1 := #alwaysON AND #State.Ready_For_Transfer;
   #_w2 := #_w1 AND #IN_Dose_Run;
   IF #_w2 THEN #State.Tank_Available := FALSE; END_IF;
   #Actuator.AV_Transfer := #_w2 AND #IN_Dose_Valve_Cmd AND #IN_Dose_LineOK;
   IF #_w1 AND #IN_FBAV_Outlet AND #IN_FBAV_Transfer AND #IN_Dose_LineOK AND #IN_FBP_Transfer AND #IN_FBCV THEN
       #State.Transfer_on_Prog := TRUE;
   END_IF;
   IF #alwaysON AND (NOT #State.Ready_For_Transfer OR (NOT #IN_Dose_Run AND NOT #IN_FBP_Transfer)) THEN
       #State.Transfer_on_Prog := FALSE;
   END_IF;
END_REGION

REGION Network 7: AV Inload
   RUNG wire#powerrail
      Contact( #alwaysON )
      wire#w1
      Contact( #Actuator.AV_Inload )
      Coil( #Out_AV_Inload )
   END_RUNG
   RUNG wire#w1
      Contact( #IN_FBAV_Inload )
      Coil( #State.Inloading )
   END_RUNG
   // the same network as SCL:
   #Out_AV_Inload := #alwaysON AND #Actuator.AV_Inload;
   #State.Inloading := #alwaysON AND #IN_FBAV_Inload;
END_REGION

REGION Network 8: AV Outlet
   RUNG wire#powerrail
      Contact( #alwaysON )
      wire#w1
      Contact( #State.Ready_For_Transfer )
      Contact( #IN_Dose_Run )
      Contact( #IN_Dose_Valve_Cmd )
      Contact( #IN_Dose_LineOK )
      Coil( #Actuator.AV_Outlet )
   END_RUNG
   RUNG wire#w1
      Contact( #Actuator.AV_Outlet )
      Coil( #Out_AV_Outlet )
   END_RUNG
   // the same network as SCL:
   #Actuator.AV_Outlet := #alwaysON AND #State.Ready_For_Transfer AND #IN_Dose_Run AND #IN_Dose_Valve_Cmd AND #IN_Dose_LineOK;
   #Out_AV_Outlet := #alwaysON AND #Actuator.AV_Outlet;
END_REGION

REGION Network 9: AV Transfer
   RUNG wire#powerrail
      Contact( #alwaysON )
      Contact( #Actuator.AV_Transfer )
      Coil( #Out_AV_Transfer )
   END_RUNG
   // the same network as SCL:
   #Out_AV_Transfer := #alwaysON AND #Actuator.AV_Transfer;
END_REGION

REGION Network 10: Pump Transfer
   RUNG wire#powerrail
      Contact( #alwaysON )
      wire#w1
      Contact( #State.Ready_For_Transfer )
      Move(in := #IN_Dose_Pump_Sp, out1 => #Out_P_Transfer_Sp)
   END_RUNG
   RUNG wire#w1
      Contact( #State.Ready_For_Transfer )
      Contact( #IN_Dose_Run )
      Contact( #IN_Dose_Pump_Cmd )
      Coil( #Actuator.P_Transfer )
   END_RUNG
   RUNG wire#w1
      Contact( #Actuator.P_Transfer )
      S_Coil( #Out_P_Transfer )
   END_RUNG
   RUNG wire#w1
      I_Contact( #Actuator.P_Transfer )
      I_Contact( #IN_FBCV )
      R_Coil( #Out_P_Transfer )
   END_RUNG
   // the same network as SCL:
   IF #alwaysON AND #State.Ready_For_Transfer THEN #Out_P_Transfer_Sp := #IN_Dose_Pump_Sp; END_IF;
   #Actuator.P_Transfer := #alwaysON AND #State.Ready_For_Transfer AND #IN_Dose_Run AND #IN_Dose_Pump_Cmd;
   IF #alwaysON AND #Actuator.P_Transfer THEN #Out_P_Transfer := TRUE; END_IF;
   IF #alwaysON AND NOT #Actuator.P_Transfer AND NOT #IN_FBCV THEN #Out_P_Transfer := FALSE; END_IF;
END_REGION

REGION Network 11: Control Valve
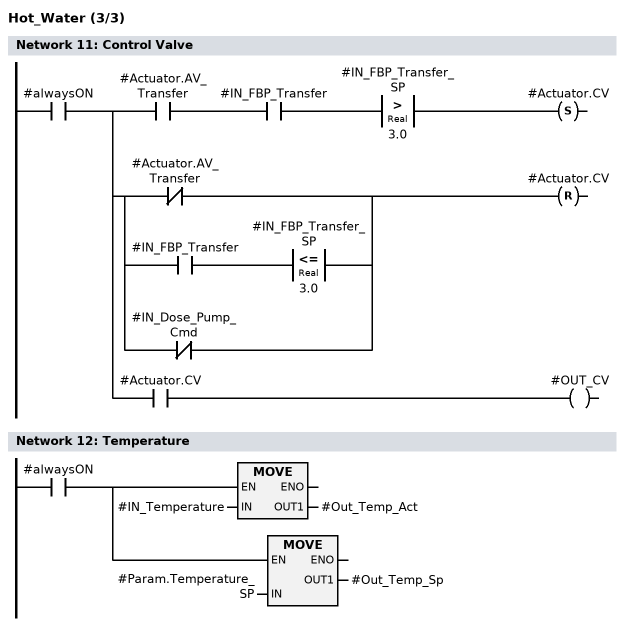
   RUNG wire#powerrail
      Contact( #alwaysON )
      wire#w1
      Contact( #Actuator.AV_Transfer )
      Contact( #IN_FBP_Transfer )
      { S7_Templates := "SrcType := Real" } GT_Contact(in1 := #IN_FBP_Transfer_SP, in2 := 3.0)
      S_Coil( #Actuator.CV )
   END_RUNG
   RUNG wire#w1
      I_Contact( #Actuator.AV_Transfer )
      wire#w2
      R_Coil( #Actuator.CV )
   END_RUNG
   RUNG wire#w1
      Contact( #IN_FBP_Transfer )
      { S7_Templates := "SrcType := Real" } LE_Contact(in1 := #IN_FBP_Transfer_SP, in2 := 3.0)
   END_RUNG wire#w2
   RUNG wire#w1
      I_Contact( #IN_Dose_Pump_Cmd )
   END_RUNG wire#w2
   RUNG wire#w1
      Contact( #Actuator.CV )
      Coil( #OUT_CV )
   END_RUNG
   // the same network as SCL:
   IF #alwaysON AND #Actuator.AV_Transfer AND #IN_FBP_Transfer AND (#IN_FBP_Transfer_SP > 3.0) THEN
       #Actuator.CV := TRUE;
   END_IF;
   IF #alwaysON AND (NOT #Actuator.AV_Transfer OR (#IN_FBP_Transfer AND (#IN_FBP_Transfer_SP <= 3.0)) OR NOT #IN_Dose_Pump_Cmd) THEN
       #Actuator.CV := FALSE;
   END_IF;
   #OUT_CV := #alwaysON AND #Actuator.CV;
END_REGION

REGION Network 12: Temperature
   RUNG wire#powerrail
      Contact( #alwaysON )
      wire#w1
      Move(in := #IN_Temperature, out1 => #Out_Temp_Act)
   END_RUNG
   RUNG wire#w1
      Move(in := #Param.Temperature_SP, out1 => #Out_Temp_Sp)
   END_RUNG
   // the same network as SCL:
   IF #alwaysON THEN
       #Out_Temp_Act := #IN_Temperature;
       #Out_Temp_Sp := #Param.Temperature_SP;
   END_IF;
END_REGION
END_FUNCTION_BLOCK

FUNCTION_BLOCK "IO Valve T02 Chili"   // FB302, LAD
{ S7_Optimized_Access := 'FALSE' }
VERSION : 0.1
// stored: AutoNumber false, IsIECCheckEnabled false, SetENOAutomatically false, UDAEnableTagReadback false
   VAR_INPUT
      lock : Bool;
      Init : Bool;
      testing : Bool;
      Reset : Bool;
   END_VAR
   VAR
      "AV-02.01" { S7_SetPoint := 'True'} : "Valve";   // AUTO BUTTERFLY VALVE INLET PROCESS WATER TO BFT CHILI AWETAN T-02.00
      "AV-02.02" { S7_SetPoint := 'True'} : "Valve";   // AUTO BUTTERFLY VALVE CIP SUPPLY TO BFT CHILI AWETAN T-02.00
      "AV-02.03" { S7_SetPoint := 'True'} : "Valve";   // AUTO BUTTERFLY VALVE OUTLET PRODUCT FROM BFT CHILI AWETAN T-02.00
      "AV-02.04" { S7_SetPoint := 'True'} : "Valve";   // AUTO BUTTERFLY VALVE OUTLET CIP TANK & LINE CHILI AWETAN T-02.00
      "AV-02.05" { S7_SetPoint := 'True'} : "Valve";   // AUTO BUTTERFLY VALVE DRAIN MONO PUMP P-02.01
      "AV-02.06" { S7_SetPoint := 'True'} : "Valve";
      "AV-02.07" { S7_SetPoint := 'True'} : "Valve";
      "AV-02.08" { S7_SetPoint := 'True'} : "Valve";
      "AV-02.09" { S7_SetPoint := 'True'} : "Valve";
      "AV-02.10" { S7_SetPoint := 'True'} : "Valve";
      "AV-02.11" { S7_SetPoint := 'True'} : "Valve";
      "AV-02.12" { S7_SetPoint := 'True'} : "Valve";
      "AV-02.13" { S7_SetPoint := 'True'} : "Valve";
      "AV-02.14" { S7_SetPoint := 'True'} : "Valve";
      "AV-02.15" { S7_SetPoint := 'True'} : "Valve";
      "AV-02.20" { S7_SetPoint := 'True'} : "Valve";
   END_VAR
BEGIN

REGION Network 1 (SCL): FB OPEN and CLOSE
   IF #testing THEN
       // Statement section IF
       #"AV-02.01".FB_OPEN := #"AV-02.01".QCMD_OP;
       #"AV-02.01".FB_CLOSE := NOT #"AV-02.01".QCMD_OP;
       #"AV-02.02".FB_OPEN := #"AV-02.02".QCMD_OP;
       #"AV-02.02".FB_CLOSE := NOT #"AV-02.02".QCMD_OP;
       #"AV-02.03".FB_OPEN := #"AV-02.03".QCMD_OP;
       #"AV-02.03".FB_CLOSE := NOT #"AV-02.03".QCMD_OP;
       #"AV-02.04".FB_OPEN := #"AV-02.04".QCMD_OP;
       #"AV-02.04".FB_CLOSE := NOT #"AV-02.04".QCMD_OP;
       #"AV-02.05".FB_OPEN := #"AV-02.05".QCMD_OP;
       #"AV-02.05".FB_CLOSE := NOT #"AV-02.05".QCMD_OP;
       #"AV-02.06".FB_OPEN := #"AV-02.06".QCMD_OP;
       #"AV-02.06".FB_CLOSE := NOT #"AV-02.06".QCMD_OP;
       #"AV-02.07".FB_OPEN := #"AV-02.07".QCMD_OP;
       #"AV-02.07".FB_CLOSE := NOT #"AV-02.07".QCMD_OP;
       #"AV-02.08".FB_OPEN := #"AV-02.08".QCMD_OP;
       #"AV-02.08".FB_CLOSE := NOT #"AV-02.08".QCMD_OP;
       #"AV-02.09".FB_OPEN := #"AV-02.09".QCMD_OP;
       #"AV-02.09".FB_CLOSE := NOT #"AV-02.09".QCMD_OP;
       #"AV-02.10".FB_OPEN := #"AV-02.10".QCMD_OP;
       #"AV-02.10".FB_CLOSE := NOT #"AV-02.10".QCMD_OP;
       #"AV-02.11".FB_OPEN := #"AV-02.11".QCMD_OP;
       #"AV-02.11".FB_CLOSE := NOT #"AV-02.11".QCMD_OP;
       #"AV-02.12".FB_OPEN := #"AV-02.12".QCMD_OP;
       #"AV-02.12".FB_CLOSE := NOT #"AV-02.12".QCMD_OP;
       #"AV-02.13".FB_OPEN := #"AV-02.13".QCMD_OP;
       #"AV-02.13".FB_CLOSE := NOT #"AV-02.13".QCMD_OP;
       #"AV-02.14".FB_OPEN := #"AV-02.14".QCMD_OP;
       #"AV-02.14".FB_CLOSE := NOT #"AV-02.14".QCMD_OP;
       #"AV-02.15".FB_OPEN := #"AV-02.15".QCMD_OP;
       #"AV-02.15".FB_CLOSE := NOT #"AV-02.15".QCMD_OP;
       #"AV-02.20".FB_OPEN := #"AV-02.20".QCMD_OP;
       #"AV-02.20".FB_CLOSE := NOT #"AV-02.20".QCMD_OP;
   ELSE
       // Statement section ELSE
       #"AV-02.01".FB_OPEN := NOT "ZSC-02.01";
       #"AV-02.01".FB_CLOSE := "ZSC-02.01";
       #"AV-02.02".FB_OPEN := NOT "ZSC-02.02";
       #"AV-02.02".FB_CLOSE := "ZSC-02.02";
       #"AV-02.03".FB_OPEN := NOT "ZSC-02.03";
       #"AV-02.03".FB_CLOSE := "ZSC-02.03";
       #"AV-02.04".FB_OPEN := NOT "ZSC-02.04";
       #"AV-02.04".FB_CLOSE := "ZSC-02.04";
       #"AV-02.05".FB_OPEN := #"AV-02.05".QCMD_OP;
       #"AV-02.05".FB_CLOSE := NOT #"AV-02.05".QCMD_OP;
       #"AV-02.06".FB_OPEN := #"AV-02.06".QCMD_OP;
       #"AV-02.06".FB_CLOSE := NOT #"AV-02.06".QCMD_OP;
       #"AV-02.07".FB_OPEN := #"AV-02.07".QCMD_OP;
       #"AV-02.07".FB_CLOSE := NOT #"AV-02.07".QCMD_OP;
       #"AV-02.08".FB_OPEN := #"AV-02.08".QCMD_OP;
       #"AV-02.08".FB_CLOSE := NOT #"AV-02.08".QCMD_OP;
       #"AV-02.09".FB_OPEN := #"AV-02.09".QCMD_OP;
       #"AV-02.09".FB_CLOSE := NOT #"AV-02.09".QCMD_OP;
       #"AV-02.10".FB_OPEN := #"AV-02.10".QCMD_OP;
       #"AV-02.10".FB_CLOSE := NOT #"AV-02.10".QCMD_OP;
       #"AV-02.11".FB_OPEN := NOT "ZSC-02.11";
       #"AV-02.11".FB_CLOSE := "ZSC-02.11";
       #"AV-02.12".FB_OPEN := NOT "ZSC-02.12";
       #"AV-02.12".FB_CLOSE := "ZSC-02.12";
       #"AV-02.13".FB_OPEN := NOT "ZSC-02.13";
       #"AV-02.13".FB_CLOSE := "ZSC-02.13";
       #"AV-02.14".FB_OPEN := #"AV-02.14".QCMD_OP;
       #"AV-02.14".FB_CLOSE := NOT #"AV-02.14".QCMD_OP;
       #"AV-02.15".FB_OPEN := #"AV-02.15".QCMD_OP;
       #"AV-02.15".FB_CLOSE := NOT #"AV-02.15".QCMD_OP;
       #"AV-02.20".FB_OPEN := #"AV-02.20".QCMD_OP;
       #"AV-02.20".FB_CLOSE := NOT #"AV-02.20".QCMD_OP;
   END_IF;
END_REGION

NETWORK
TITLE = FB Monitoring Time
// FB OPEN Time
      L     t#20s;
      T     #"AV-02.01".MON_T;
      T     #"AV-02.02".MON_T;
      T     #"AV-02.03".MON_T;
      T     #"AV-02.04".MON_T;
      T     #"AV-02.05".MON_T;
      T     #"AV-02.06".MON_T;
      T     #"AV-02.07".MON_T;
      T     #"AV-02.08".MON_T;
      T     #"AV-02.09".MON_T;
      T     #"AV-02.10".MON_T;
      T     #"AV-02.11".MON_T;
      T     #"AV-02.12".MON_T;
      T     #"AV-02.13".MON_T;
      T     #"AV-02.14".MON_T;
      T     #"AV-02.15".MON_T;
      T     #"AV-02.20".MON_T;
// FB CLOSE Time
      L     t#20s;
      T     #"AV-02.01".MON_T_CLOSE;
      T     #"AV-02.02".MON_T_CLOSE;
      T     #"AV-02.03".MON_T_CLOSE;
      T     #"AV-02.04".MON_T_CLOSE;
      T     #"AV-02.05".MON_T_CLOSE;
      T     #"AV-02.06".MON_T_CLOSE;
      T     #"AV-02.07".MON_T_CLOSE;
      T     #"AV-02.08".MON_T_CLOSE;
      T     #"AV-02.09".MON_T_CLOSE;
      T     #"AV-02.10".MON_T_CLOSE;
      T     #"AV-02.11".MON_T_CLOSE;
      T     #"AV-02.12".MON_T_CLOSE;
      T     #"AV-02.13".MON_T_CLOSE;
      T     #"AV-02.14".MON_T_CLOSE;
      T     #"AV-02.15".MON_T_CLOSE;
      T     #"AV-02.20".MON_T_CLOSE;

REGION Network 3: AV-02.01 w ZSC
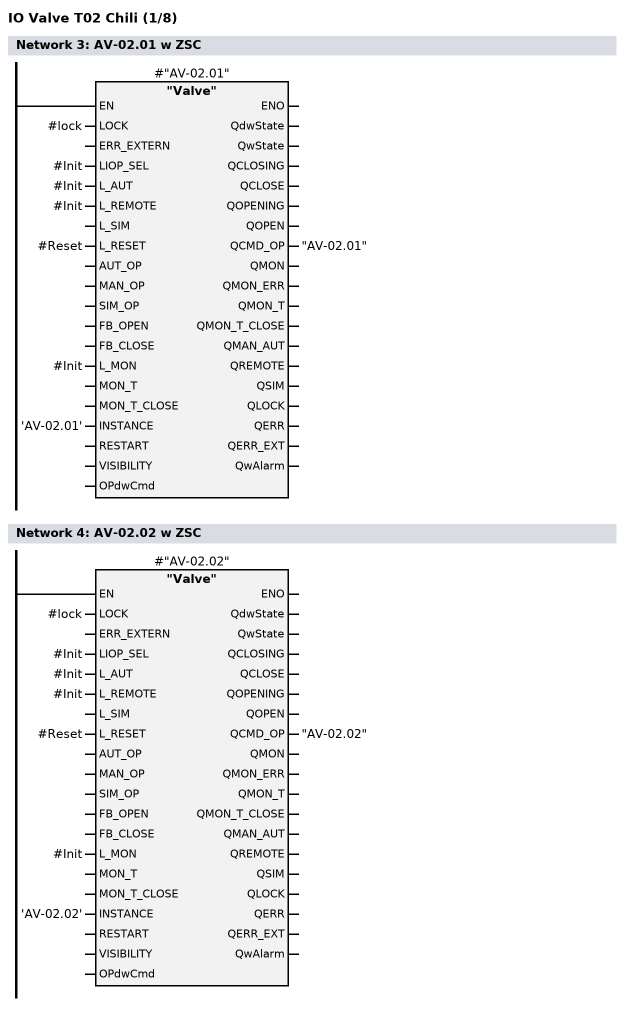
   RUNG wire#powerrail
      #"AV-02.01"(LOCK := #lock, ERR_EXTERN :=, LIOP_SEL := #Init, L_AUT := #Init, L_REMOTE := #Init, L_SIM :=, L_RESET := #Reset, AUT_OP :=, MAN_OP :=, SIM_OP :=, FB_OPEN :=, FB_CLOSE :=, L_MON := #Init, MON_T :=, MON_T_CLOSE :=, INSTANCE := 'AV-02.01', RESTART :=, VISIBILITY :=, OPdwCmd :=, QdwState =>, QwState =>, QCLOSING =>, QCLOSE =>, QOPENING =>, QOPEN =>, QCMD_OP => "AV-02.01", QMON =>, QMON_ERR =>, QMON_T =>, QMON_T_CLOSE =>, QMAN_AUT =>, QREMOTE =>, QSIM =>, QLOCK =>, QERR =>, QERR_EXT =>, QwAlarm =>)
   END_RUNG
   // the same network as SCL:
   #"AV-02.01"(LOCK := #lock,   // "Valve"
               LIOP_SEL := #Init,
               L_AUT := #Init,
               L_REMOTE := #Init,
               L_RESET := #Reset,
               L_MON := #Init,
               INSTANCE := 'AV-02.01',
               QCMD_OP => "AV-02.01");
END_REGION

REGION Network 4: AV-02.02 w ZSC
   RUNG wire#powerrail
      #"AV-02.02"(LOCK := #lock, ERR_EXTERN :=, LIOP_SEL := #Init, L_AUT := #Init, L_REMOTE := #Init, L_SIM :=, L_RESET := #Reset, AUT_OP :=, MAN_OP :=, SIM_OP :=, FB_OPEN :=, FB_CLOSE :=, L_MON := #Init, MON_T :=, MON_T_CLOSE :=, INSTANCE := 'AV-02.02', RESTART :=, VISIBILITY :=, OPdwCmd :=, QdwState =>, QwState =>, QCLOSING =>, QCLOSE =>, QOPENING =>, QOPEN =>, QCMD_OP => "AV-02.02", QMON =>, QMON_ERR =>, QMON_T =>, QMON_T_CLOSE =>, QMAN_AUT =>, QREMOTE =>, QSIM =>, QLOCK =>, QERR =>, QERR_EXT =>, QwAlarm =>)
   END_RUNG
   // the same network as SCL:
   #"AV-02.02"(LOCK := #lock,   // "Valve"
               LIOP_SEL := #Init,
               L_AUT := #Init,
               L_REMOTE := #Init,
               L_RESET := #Reset,
               L_MON := #Init,
               INSTANCE := 'AV-02.02',
               QCMD_OP => "AV-02.02");
END_REGION

REGION Network 5: AV-02.03 w ZSC
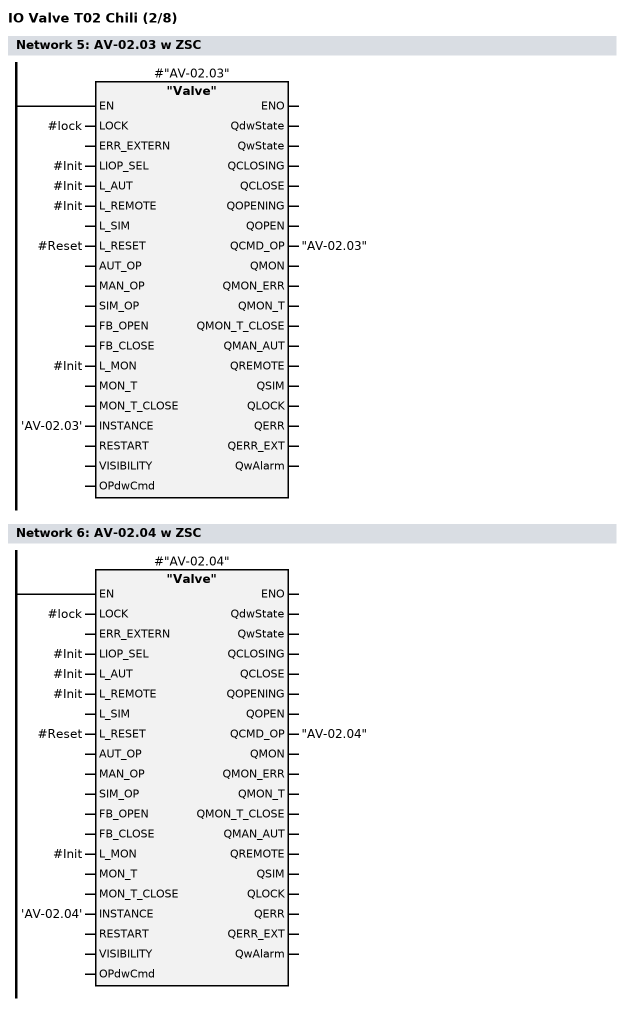
   RUNG wire#powerrail
      #"AV-02.03"(LOCK := #lock, ERR_EXTERN :=, LIOP_SEL := #Init, L_AUT := #Init, L_REMOTE := #Init, L_SIM :=, L_RESET := #Reset, AUT_OP :=, MAN_OP :=, SIM_OP :=, FB_OPEN :=, FB_CLOSE :=, L_MON := #Init, MON_T :=, MON_T_CLOSE :=, INSTANCE := 'AV-02.03', RESTART :=, VISIBILITY :=, OPdwCmd :=, QdwState =>, QwState =>, QCLOSING =>, QCLOSE =>, QOPENING =>, QOPEN =>, QCMD_OP => "AV-02.03", QMON =>, QMON_ERR =>, QMON_T =>, QMON_T_CLOSE =>, QMAN_AUT =>, QREMOTE =>, QSIM =>, QLOCK =>, QERR =>, QERR_EXT =>, QwAlarm =>)
   END_RUNG
   // the same network as SCL:
   #"AV-02.03"(LOCK := #lock,   // "Valve"
               LIOP_SEL := #Init,
               L_AUT := #Init,
               L_REMOTE := #Init,
               L_RESET := #Reset,
               L_MON := #Init,
               INSTANCE := 'AV-02.03',
               QCMD_OP => "AV-02.03");
END_REGION

REGION Network 6: AV-02.04 w ZSC
   RUNG wire#powerrail
      #"AV-02.04"(LOCK := #lock, ERR_EXTERN :=, LIOP_SEL := #Init, L_AUT := #Init, L_REMOTE := #Init, L_SIM :=, L_RESET := #Reset, AUT_OP :=, MAN_OP :=, SIM_OP :=, FB_OPEN :=, FB_CLOSE :=, L_MON := #Init, MON_T :=, MON_T_CLOSE :=, INSTANCE := 'AV-02.04', RESTART :=, VISIBILITY :=, OPdwCmd :=, QdwState =>, QwState =>, QCLOSING =>, QCLOSE =>, QOPENING =>, QOPEN =>, QCMD_OP => "AV-02.04", QMON =>, QMON_ERR =>, QMON_T =>, QMON_T_CLOSE =>, QMAN_AUT =>, QREMOTE =>, QSIM =>, QLOCK =>, QERR =>, QERR_EXT =>, QwAlarm =>)
   END_RUNG
   // the same network as SCL:
   #"AV-02.04"(LOCK := #lock,   // "Valve"
               LIOP_SEL := #Init,
               L_AUT := #Init,
               L_REMOTE := #Init,
               L_RESET := #Reset,
               L_MON := #Init,
               INSTANCE := 'AV-02.04',
               QCMD_OP => "AV-02.04");
END_REGION

REGION Network 7: AV-02.05
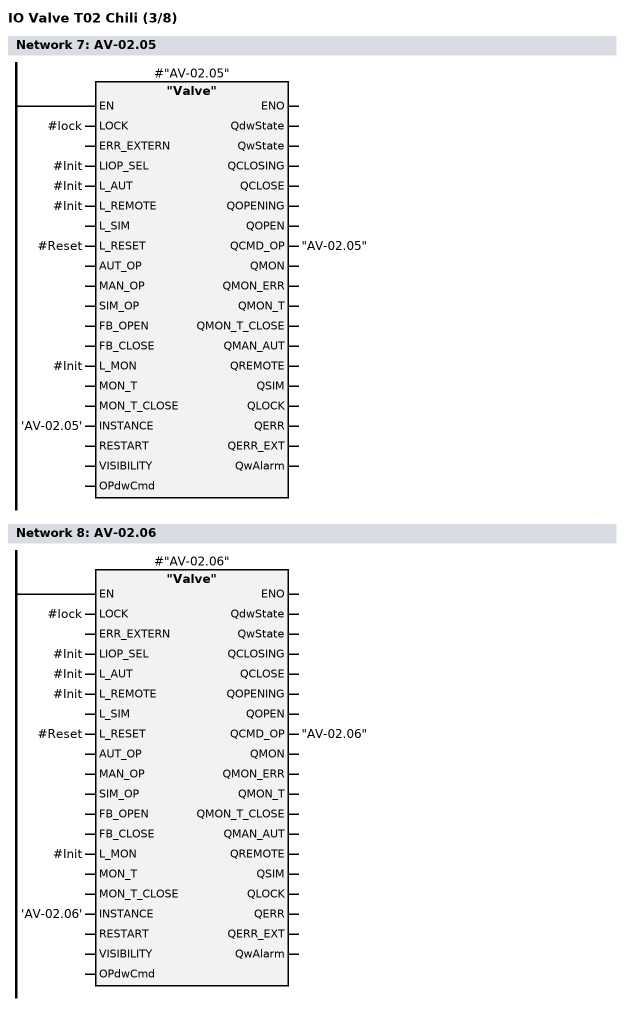
   RUNG wire#powerrail
      #"AV-02.05"(LOCK := #lock, ERR_EXTERN :=, LIOP_SEL := #Init, L_AUT := #Init, L_REMOTE := #Init, L_SIM :=, L_RESET := #Reset, AUT_OP :=, MAN_OP :=, SIM_OP :=, FB_OPEN :=, FB_CLOSE :=, L_MON := #Init, MON_T :=, MON_T_CLOSE :=, INSTANCE := 'AV-02.05', RESTART :=, VISIBILITY :=, OPdwCmd :=, QdwState =>, QwState =>, QCLOSING =>, QCLOSE =>, QOPENING =>, QOPEN =>, QCMD_OP => "AV-02.05", QMON =>, QMON_ERR =>, QMON_T =>, QMON_T_CLOSE =>, QMAN_AUT =>, QREMOTE =>, QSIM =>, QLOCK =>, QERR =>, QERR_EXT =>, QwAlarm =>)
   END_RUNG
   // the same network as SCL:
   #"AV-02.05"(LOCK := #lock,   // "Valve"
               LIOP_SEL := #Init,
               L_AUT := #Init,
               L_REMOTE := #Init,
               L_RESET := #Reset,
               L_MON := #Init,
               INSTANCE := 'AV-02.05',
               QCMD_OP => "AV-02.05");
END_REGION

REGION Network 8: AV-02.06
   RUNG wire#powerrail
      #"AV-02.06"(LOCK := #lock, ERR_EXTERN :=, LIOP_SEL := #Init, L_AUT := #Init, L_REMOTE := #Init, L_SIM :=, L_RESET := #Reset, AUT_OP :=, MAN_OP :=, SIM_OP :=, FB_OPEN :=, FB_CLOSE :=, L_MON := #Init, MON_T :=, MON_T_CLOSE :=, INSTANCE := 'AV-02.06', RESTART :=, VISIBILITY :=, OPdwCmd :=, QdwState =>, QwState =>, QCLOSING =>, QCLOSE =>, QOPENING =>, QOPEN =>, QCMD_OP => "AV-02.06", QMON =>, QMON_ERR =>, QMON_T =>, QMON_T_CLOSE =>, QMAN_AUT =>, QREMOTE =>, QSIM =>, QLOCK =>, QERR =>, QERR_EXT =>, QwAlarm =>)
   END_RUNG
   // the same network as SCL:
   #"AV-02.06"(LOCK := #lock,   // "Valve"
               LIOP_SEL := #Init,
               L_AUT := #Init,
               L_REMOTE := #Init,
               L_RESET := #Reset,
               L_MON := #Init,
               INSTANCE := 'AV-02.06',
               QCMD_OP => "AV-02.06");
END_REGION

REGION Network 9: AV-02.07
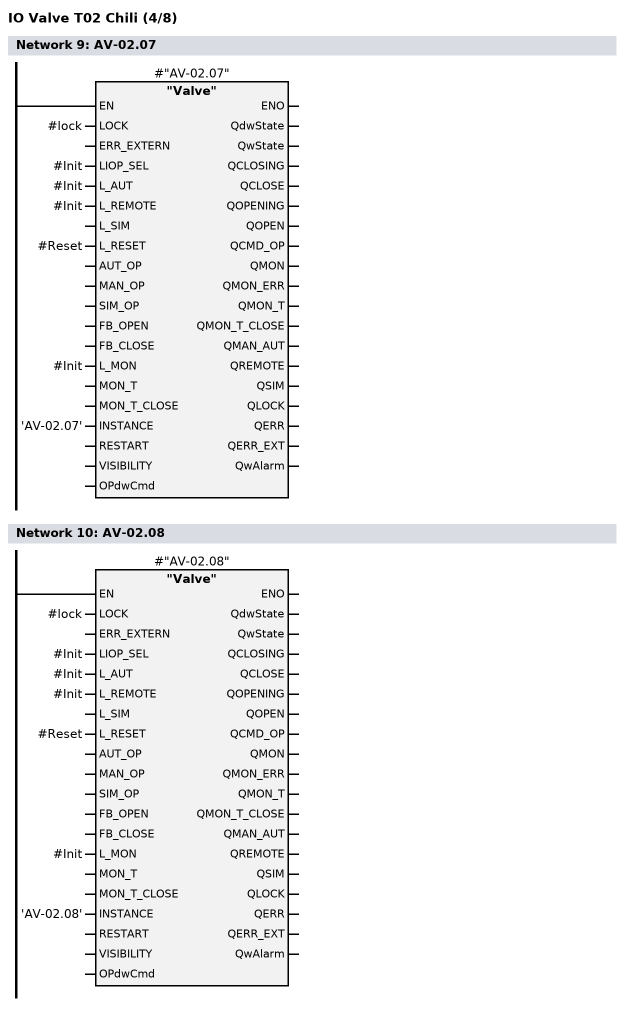
   RUNG wire#powerrail
      #"AV-02.07"(LOCK := #lock, ERR_EXTERN :=, LIOP_SEL := #Init, L_AUT := #Init, L_REMOTE := #Init, L_SIM :=, L_RESET := #Reset, AUT_OP :=, MAN_OP :=, SIM_OP :=, FB_OPEN :=, FB_CLOSE :=, L_MON := #Init, MON_T :=, MON_T_CLOSE :=, INSTANCE := 'AV-02.07', RESTART :=, VISIBILITY :=, OPdwCmd :=, QdwState =>, QwState =>, QCLOSING =>, QCLOSE =>, QOPENING =>, QOPEN =>, QCMD_OP =>, QMON =>, QMON_ERR =>, QMON_T =>, QMON_T_CLOSE =>, QMAN_AUT =>, QREMOTE =>, QSIM =>, QLOCK =>, QERR =>, QERR_EXT =>, QwAlarm =>)
   END_RUNG
   // the same network as SCL:
   #"AV-02.07"(LOCK := #lock,   // "Valve"
               LIOP_SEL := #Init,
               L_AUT := #Init,
               L_REMOTE := #Init,
               L_RESET := #Reset,
               L_MON := #Init,
               INSTANCE := 'AV-02.07');
END_REGION

REGION Network 10: AV-02.08
   RUNG wire#powerrail
      #"AV-02.08"(LOCK := #lock, ERR_EXTERN :=, LIOP_SEL := #Init, L_AUT := #Init, L_REMOTE := #Init, L_SIM :=, L_RESET := #Reset, AUT_OP :=, MAN_OP :=, SIM_OP :=, FB_OPEN :=, FB_CLOSE :=, L_MON := #Init, MON_T :=, MON_T_CLOSE :=, INSTANCE := 'AV-02.08', RESTART :=, VISIBILITY :=, OPdwCmd :=, QdwState =>, QwState =>, QCLOSING =>, QCLOSE =>, QOPENING =>, QOPEN =>, QCMD_OP =>, QMON =>, QMON_ERR =>, QMON_T =>, QMON_T_CLOSE =>, QMAN_AUT =>, QREMOTE =>, QSIM =>, QLOCK =>, QERR =>, QERR_EXT =>, QwAlarm =>)
   END_RUNG
   // the same network as SCL:
   #"AV-02.08"(LOCK := #lock,   // "Valve"
               LIOP_SEL := #Init,
               L_AUT := #Init,
               L_REMOTE := #Init,
               L_RESET := #Reset,
               L_MON := #Init,
               INSTANCE := 'AV-02.08');
END_REGION

REGION Network 11: AV-02.09
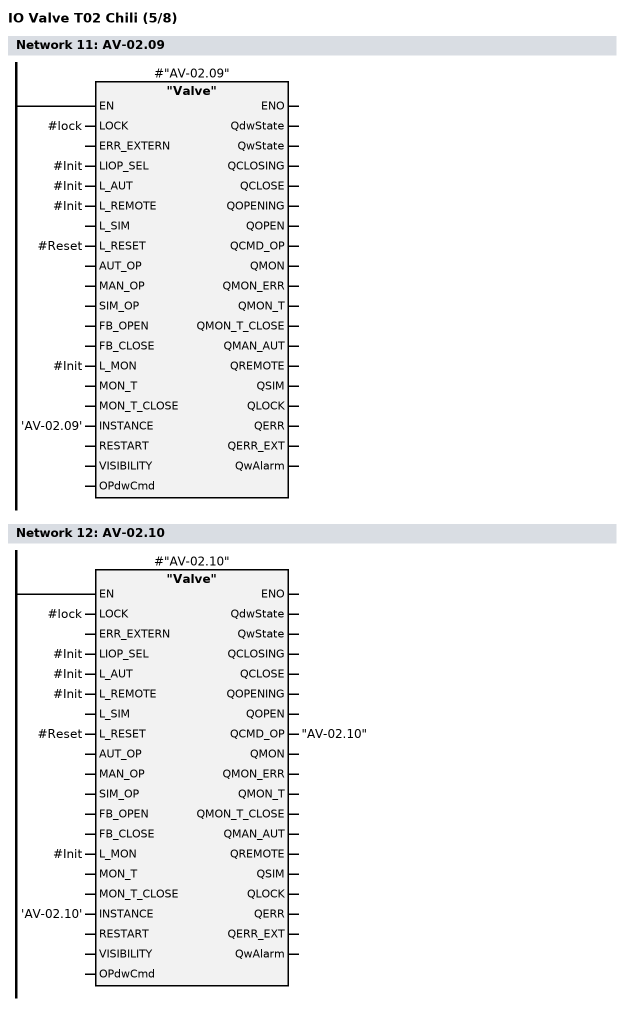
   RUNG wire#powerrail
      #"AV-02.09"(LOCK := #lock, ERR_EXTERN :=, LIOP_SEL := #Init, L_AUT := #Init, L_REMOTE := #Init, L_SIM :=, L_RESET := #Reset, AUT_OP :=, MAN_OP :=, SIM_OP :=, FB_OPEN :=, FB_CLOSE :=, L_MON := #Init, MON_T :=, MON_T_CLOSE :=, INSTANCE := 'AV-02.09', RESTART :=, VISIBILITY :=, OPdwCmd :=, QdwState =>, QwState =>, QCLOSING =>, QCLOSE =>, QOPENING =>, QOPEN =>, QCMD_OP =>, QMON =>, QMON_ERR =>, QMON_T =>, QMON_T_CLOSE =>, QMAN_AUT =>, QREMOTE =>, QSIM =>, QLOCK =>, QERR =>, QERR_EXT =>, QwAlarm =>)
   END_RUNG
   // the same network as SCL:
   #"AV-02.09"(LOCK := #lock,   // "Valve"
               LIOP_SEL := #Init,
               L_AUT := #Init,
               L_REMOTE := #Init,
               L_RESET := #Reset,
               L_MON := #Init,
               INSTANCE := 'AV-02.09');
END_REGION

REGION Network 12: AV-02.10
   RUNG wire#powerrail
      #"AV-02.10"(LOCK := #lock, ERR_EXTERN :=, LIOP_SEL := #Init, L_AUT := #Init, L_REMOTE := #Init, L_SIM :=, L_RESET := #Reset, AUT_OP :=, MAN_OP :=, SIM_OP :=, FB_OPEN :=, FB_CLOSE :=, L_MON := #Init, MON_T :=, MON_T_CLOSE :=, INSTANCE := 'AV-02.10', RESTART :=, VISIBILITY :=, OPdwCmd :=, QdwState =>, QwState =>, QCLOSING =>, QCLOSE =>, QOPENING =>, QOPEN =>, QCMD_OP => "AV-02.10", QMON =>, QMON_ERR =>, QMON_T =>, QMON_T_CLOSE =>, QMAN_AUT =>, QREMOTE =>, QSIM =>, QLOCK =>, QERR =>, QERR_EXT =>, QwAlarm =>)
   END_RUNG
   // the same network as SCL:
   #"AV-02.10"(LOCK := #lock,   // "Valve"
               LIOP_SEL := #Init,
               L_AUT := #Init,
               L_REMOTE := #Init,
               L_RESET := #Reset,
               L_MON := #Init,
               INSTANCE := 'AV-02.10',
               QCMD_OP => "AV-02.10");
END_REGION

REGION Network 13: AV-02.11 w ZSC
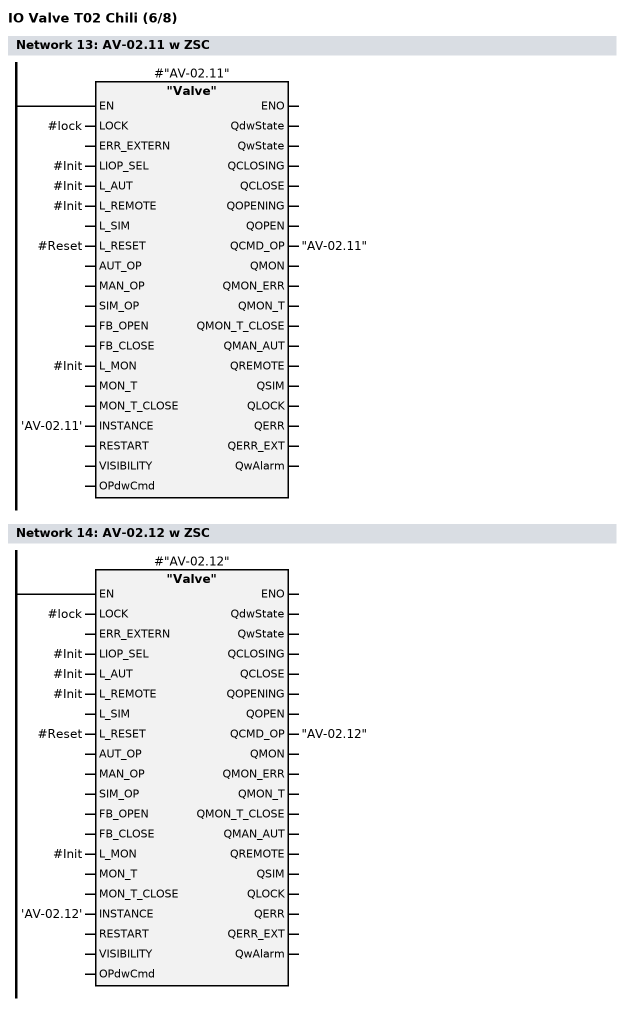
   RUNG wire#powerrail
      #"AV-02.11"(LOCK := #lock, ERR_EXTERN :=, LIOP_SEL := #Init, L_AUT := #Init, L_REMOTE := #Init, L_SIM :=, L_RESET := #Reset, AUT_OP :=, MAN_OP :=, SIM_OP :=, FB_OPEN :=, FB_CLOSE :=, L_MON := #Init, MON_T :=, MON_T_CLOSE :=, INSTANCE := 'AV-02.11', RESTART :=, VISIBILITY :=, OPdwCmd :=, QdwState =>, QwState =>, QCLOSING =>, QCLOSE =>, QOPENING =>, QOPEN =>, QCMD_OP => "AV-02.11", QMON =>, QMON_ERR =>, QMON_T =>, QMON_T_CLOSE =>, QMAN_AUT =>, QREMOTE =>, QSIM =>, QLOCK =>, QERR =>, QERR_EXT =>, QwAlarm =>)
   END_RUNG
   // the same network as SCL:
   #"AV-02.11"(LOCK := #lock,   // "Valve"
               LIOP_SEL := #Init,
               L_AUT := #Init,
               L_REMOTE := #Init,
               L_RESET := #Reset,
               L_MON := #Init,
               INSTANCE := 'AV-02.11',
               QCMD_OP => "AV-02.11");
END_REGION

REGION Network 14: AV-02.12 w ZSC
   RUNG wire#powerrail
      #"AV-02.12"(LOCK := #lock, ERR_EXTERN :=, LIOP_SEL := #Init, L_AUT := #Init, L_REMOTE := #Init, L_SIM :=, L_RESET := #Reset, AUT_OP :=, MAN_OP :=, SIM_OP :=, FB_OPEN :=, FB_CLOSE :=, L_MON := #Init, MON_T :=, MON_T_CLOSE :=, INSTANCE := 'AV-02.12', RESTART :=, VISIBILITY :=, OPdwCmd :=, QdwState =>, QwState =>, QCLOSING =>, QCLOSE =>, QOPENING =>, QOPEN =>, QCMD_OP => "AV-02.12", QMON =>, QMON_ERR =>, QMON_T =>, QMON_T_CLOSE =>, QMAN_AUT =>, QREMOTE =>, QSIM =>, QLOCK =>, QERR =>, QERR_EXT =>, QwAlarm =>)
   END_RUNG
   // the same network as SCL:
   #"AV-02.12"(LOCK := #lock,   // "Valve"
               LIOP_SEL := #Init,
               L_AUT := #Init,
               L_REMOTE := #Init,
               L_RESET := #Reset,
               L_MON := #Init,
               INSTANCE := 'AV-02.12',
               QCMD_OP => "AV-02.12");
END_REGION

REGION Network 15: AV-02.13 w ZSC
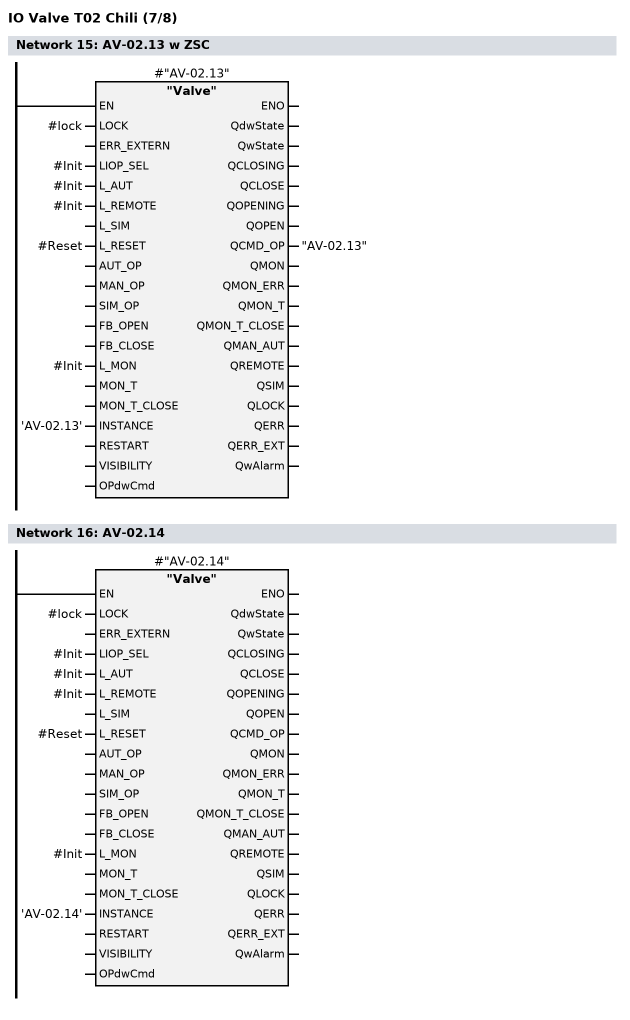
   RUNG wire#powerrail
      #"AV-02.13"(LOCK := #lock, ERR_EXTERN :=, LIOP_SEL := #Init, L_AUT := #Init, L_REMOTE := #Init, L_SIM :=, L_RESET := #Reset, AUT_OP :=, MAN_OP :=, SIM_OP :=, FB_OPEN :=, FB_CLOSE :=, L_MON := #Init, MON_T :=, MON_T_CLOSE :=, INSTANCE := 'AV-02.13', RESTART :=, VISIBILITY :=, OPdwCmd :=, QdwState =>, QwState =>, QCLOSING =>, QCLOSE =>, QOPENING =>, QOPEN =>, QCMD_OP => "AV-02.13", QMON =>, QMON_ERR =>, QMON_T =>, QMON_T_CLOSE =>, QMAN_AUT =>, QREMOTE =>, QSIM =>, QLOCK =>, QERR =>, QERR_EXT =>, QwAlarm =>)
   END_RUNG
   // the same network as SCL:
   #"AV-02.13"(LOCK := #lock,   // "Valve"
               LIOP_SEL := #Init,
               L_AUT := #Init,
               L_REMOTE := #Init,
               L_RESET := #Reset,
               L_MON := #Init,
               INSTANCE := 'AV-02.13',
               QCMD_OP => "AV-02.13");
END_REGION

REGION Network 16: AV-02.14
   RUNG wire#powerrail
      #"AV-02.14"(LOCK := #lock, ERR_EXTERN :=, LIOP_SEL := #Init, L_AUT := #Init, L_REMOTE := #Init, L_SIM :=, L_RESET := #Reset, AUT_OP :=, MAN_OP :=, SIM_OP :=, FB_OPEN :=, FB_CLOSE :=, L_MON := #Init, MON_T :=, MON_T_CLOSE :=, INSTANCE := 'AV-02.14', RESTART :=, VISIBILITY :=, OPdwCmd :=, QdwState =>, QwState =>, QCLOSING =>, QCLOSE =>, QOPENING =>, QOPEN =>, QCMD_OP =>, QMON =>, QMON_ERR =>, QMON_T =>, QMON_T_CLOSE =>, QMAN_AUT =>, QREMOTE =>, QSIM =>, QLOCK =>, QERR =>, QERR_EXT =>, QwAlarm =>)
   END_RUNG
   // the same network as SCL:
   #"AV-02.14"(LOCK := #lock,   // "Valve"
               LIOP_SEL := #Init,
               L_AUT := #Init,
               L_REMOTE := #Init,
               L_RESET := #Reset,
               L_MON := #Init,
               INSTANCE := 'AV-02.14');
END_REGION

REGION Network 17: AV-02.15
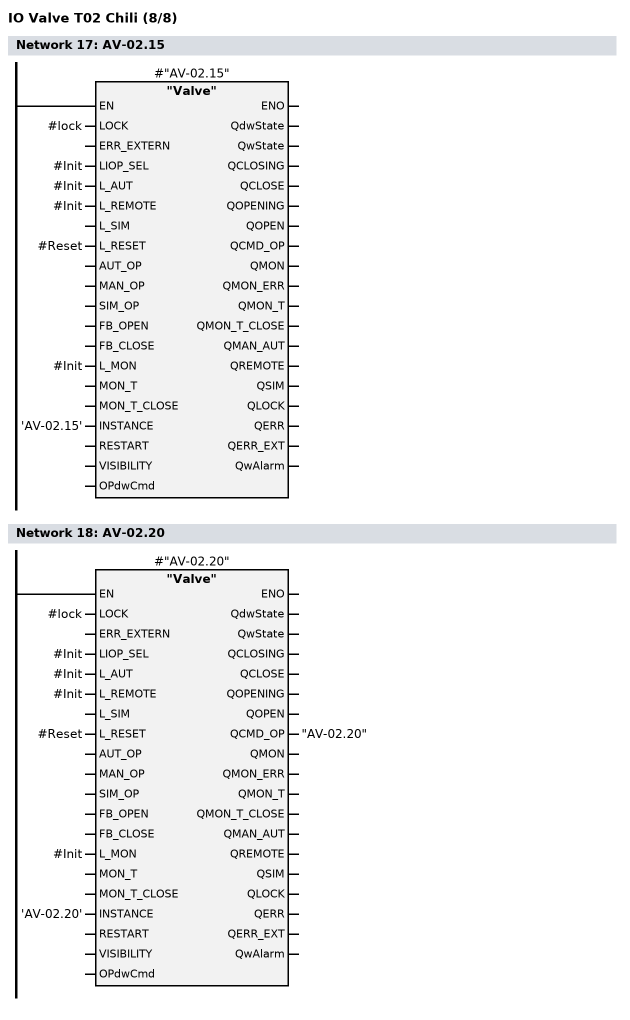
   RUNG wire#powerrail
      #"AV-02.15"(LOCK := #lock, ERR_EXTERN :=, LIOP_SEL := #Init, L_AUT := #Init, L_REMOTE := #Init, L_SIM :=, L_RESET := #Reset, AUT_OP :=, MAN_OP :=, SIM_OP :=, FB_OPEN :=, FB_CLOSE :=, L_MON := #Init, MON_T :=, MON_T_CLOSE :=, INSTANCE := 'AV-02.15', RESTART :=, VISIBILITY :=, OPdwCmd :=, QdwState =>, QwState =>, QCLOSING =>, QCLOSE =>, QOPENING =>, QOPEN =>, QCMD_OP =>, QMON =>, QMON_ERR =>, QMON_T =>, QMON_T_CLOSE =>, QMAN_AUT =>, QREMOTE =>, QSIM =>, QLOCK =>, QERR =>, QERR_EXT =>, QwAlarm =>)
   END_RUNG
   // the same network as SCL:
   #"AV-02.15"(LOCK := #lock,   // "Valve"
               LIOP_SEL := #Init,
               L_AUT := #Init,
               L_REMOTE := #Init,
               L_RESET := #Reset,
               L_MON := #Init,
               INSTANCE := 'AV-02.15');
END_REGION

REGION Network 18: AV-02.20
   RUNG wire#powerrail
      #"AV-02.20"(LOCK := #lock, ERR_EXTERN :=, LIOP_SEL := #Init, L_AUT := #Init, L_REMOTE := #Init, L_SIM :=, L_RESET := #Reset, AUT_OP :=, MAN_OP :=, SIM_OP :=, FB_OPEN :=, FB_CLOSE :=, L_MON := #Init, MON_T :=, MON_T_CLOSE :=, INSTANCE := 'AV-02.20', RESTART :=, VISIBILITY :=, OPdwCmd :=, QdwState =>, QwState =>, QCLOSING =>, QCLOSE =>, QOPENING =>, QOPEN =>, QCMD_OP => "AV-02.20", QMON =>, QMON_ERR =>, QMON_T =>, QMON_T_CLOSE =>, QMAN_AUT =>, QREMOTE =>, QSIM =>, QLOCK =>, QERR =>, QERR_EXT =>, QwAlarm =>)
   END_RUNG
   // the same network as SCL:
   #"AV-02.20"(LOCK := #lock,   // "Valve"
               LIOP_SEL := #Init,
               L_AUT := #Init,
               L_REMOTE := #Init,
               L_RESET := #Reset,
               L_MON := #Init,
               INSTANCE := 'AV-02.20',
               QCMD_OP => "AV-02.20");
END_REGION
END_FUNCTION_BLOCK

FUNCTION_BLOCK "IO Valve T03 Chili"   // FB303, LAD
{ S7_Optimized_Access := 'FALSE' }
VERSION : 0.1
// stored: AutoNumber false, IsIECCheckEnabled false, SetENOAutomatically false, UDAEnableTagReadback false
   VAR_INPUT
      lock : Bool;
      Init : Bool;
      testing : Bool;
      Reset : Bool;
   END_VAR
   VAR
      "AV-03.01" { S7_SetPoint := 'True'} : "Valve";   // AUTO BUTTERFLY VALVE INLET PROCESS WATER TO BFT CHILI AWETAN T-03.00
      "AV-03.02" { S7_SetPoint := 'True'} : "Valve";   // AUTO BUTTERFLY VALVE CIP SUPPLY TO BFT CHILI AWETAN T-03.00
      "AV-03.03" { S7_SetPoint := 'True'} : "Valve";   // AUTO BUTTERFLY VALVE OUTLET PRODUCT FROM BFT CHILI AWETAN T-03.00
      "AV-03.04" { S7_SetPoint := 'True'} : "Valve";   // AUTO BUTTERFLY VALVE OUTLET CIP TANK & LINE CHILI AWETAN T-03.00
      "AV-03.05" { S7_SetPoint := 'True'} : "Valve";   // AUTO BUTTERFLY VALVE DRAIN MONO PUMP P-03.01
      "AV-03.06" { S7_SetPoint := 'True'} : "Valve";   // AUTO BUTTERFLY VALVE INLET PRODUCT TO BFT CHILI AWETAN T-03.00
      "AV-03.07" { S7_SetPoint := 'True'} : "Valve";   // AUTO BUTTERFLY VALVE INLET CHILI AWETAN FROM T-02.00 TO BLENDING TANK T-20.00
      "AV-03.08" { S7_SetPoint := 'True'} : "Valve";
      "AV-03.09" { S7_SetPoint := 'True'} : "Valve";
      "AV-03.10" { S7_SetPoint := 'True'} : "Valve";
      "AV-03.11" { S7_SetPoint := 'True'} : "Valve";
      "AV-03.12" { S7_SetPoint := 'True'} : "Valve";
      "AV-03.13" { S7_SetPoint := 'True'} : "Valve";
      "AV-03.14" { S7_SetPoint := 'True'} : "Valve";
      "AV-03.15" { S7_SetPoint := 'True'} : "Valve";
   END_VAR
BEGIN

REGION Network 1 (SCL): FB OPEN and CLOSE
   IF #testing THEN
       // Statement section IF
       #"AV-03.01".FB_OPEN := #"AV-03.01".QCMD_OP;
       #"AV-03.01".FB_CLOSE := NOT #"AV-03.01".QCMD_OP;
       #"AV-03.02".FB_OPEN := #"AV-03.02".QCMD_OP;
       #"AV-03.02".FB_CLOSE := NOT #"AV-03.02".QCMD_OP;
       #"AV-03.03".FB_OPEN := #"AV-03.03".QCMD_OP;
       #"AV-03.03".FB_CLOSE := NOT #"AV-03.03".QCMD_OP;
       #"AV-03.04".FB_OPEN := #"AV-03.04".QCMD_OP;
       #"AV-03.04".FB_CLOSE := NOT #"AV-03.04".QCMD_OP;
       #"AV-03.05".FB_OPEN := #"AV-03.05".QCMD_OP;
       #"AV-03.05".FB_CLOSE := NOT #"AV-03.05".QCMD_OP;
       #"AV-03.06".FB_OPEN := #"AV-03.06".QCMD_OP;
       #"AV-03.06".FB_CLOSE := NOT #"AV-03.06".QCMD_OP;
       #"AV-03.07".FB_OPEN := #"AV-03.07".QCMD_OP;
       #"AV-03.07".FB_CLOSE := NOT #"AV-03.07".QCMD_OP;
       #"AV-03.08".FB_OPEN := #"AV-03.08".QCMD_OP;
       #"AV-03.08".FB_CLOSE := NOT #"AV-03.08".QCMD_OP;
       #"AV-03.09".FB_OPEN := #"AV-03.09".QCMD_OP;
       #"AV-03.09".FB_CLOSE := NOT #"AV-03.09".QCMD_OP;
       #"AV-03.10".FB_OPEN := #"AV-03.10".QCMD_OP;
       #"AV-03.10".FB_CLOSE := NOT #"AV-03.10".QCMD_OP;
       #"AV-03.11".FB_OPEN := #"AV-03.11".QCMD_OP;
       #"AV-03.11".FB_CLOSE := NOT #"AV-03.11".QCMD_OP;
       #"AV-03.12".FB_OPEN := #"AV-03.12".QCMD_OP;
       #"AV-03.12".FB_CLOSE := NOT #"AV-03.12".QCMD_OP;
       #"AV-03.13".FB_OPEN := #"AV-03.13".QCMD_OP;
       #"AV-03.13".FB_CLOSE := NOT #"AV-03.13".QCMD_OP;
       #"AV-03.14".FB_OPEN := #"AV-03.14".QCMD_OP;
       #"AV-03.14".FB_CLOSE := NOT #"AV-03.14".QCMD_OP;
       #"AV-03.15".FB_OPEN := #"AV-03.15".QCMD_OP;
       #"AV-03.15".FB_CLOSE := NOT #"AV-03.15".QCMD_OP;
   ELSE
       // Statement section ELSE
       #"AV-03.01".FB_OPEN := NOT "ZSC-03.01";
       #"AV-03.01".FB_CLOSE := "ZSC-03.01";
       #"AV-03.02".FB_OPEN := NOT "ZSC-03.02";
       #"AV-03.02".FB_CLOSE := "ZSC-03.02";
       #"AV-03.03".FB_OPEN := NOT "ZSC-03.03";
       #"AV-03.03".FB_CLOSE := "ZSC-03.03";
       #"AV-03.04".FB_OPEN := NOT "ZSC-03.04";
       #"AV-03.04".FB_CLOSE := "ZSC-03.04";
       #"AV-03.05".FB_OPEN := #"AV-03.05".QCMD_OP;
       #"AV-03.05".FB_CLOSE := NOT #"AV-03.05".QCMD_OP;
       #"AV-03.06".FB_OPEN := NOT "ZSC-03.06";
       #"AV-03.06".FB_CLOSE := "ZSC-03.06";
       #"AV-03.07".FB_OPEN := #"AV-03.07".QCMD_OP;
       #"AV-03.07".FB_CLOSE := NOT #"AV-03.07".QCMD_OP;
       #"AV-03.08".FB_OPEN := #"AV-03.08".QCMD_OP;
       #"AV-03.08".FB_CLOSE := NOT #"AV-03.08".QCMD_OP;
       #"AV-03.09".FB_OPEN := #"AV-03.09".QCMD_OP;
       #"AV-03.09".FB_CLOSE := NOT #"AV-03.09".QCMD_OP;
       #"AV-03.10".FB_OPEN := #"AV-03.10".QCMD_OP;
       #"AV-03.10".FB_CLOSE := NOT #"AV-03.10".QCMD_OP;
       #"AV-03.11".FB_OPEN := NOT "ZSC-03.11";
       #"AV-03.11".FB_CLOSE := "ZSC-03.11";
       #"AV-03.12".FB_OPEN := NOT "ZSC-03.12";
       #"AV-03.12".FB_CLOSE := "ZSC-03.12";
       #"AV-03.13".FB_OPEN := NOT "ZSC-03.13";
       #"AV-03.13".FB_CLOSE := "ZSC-03.13";
       #"AV-03.14".FB_OPEN := #"AV-03.14".QCMD_OP;
       #"AV-03.14".FB_CLOSE := NOT #"AV-03.14".QCMD_OP;
       #"AV-03.15".FB_OPEN := #"AV-03.15".QCMD_OP;
       #"AV-03.15".FB_CLOSE := NOT #"AV-03.15".QCMD_OP;
   END_IF;
END_REGION

NETWORK
TITLE = FB Monitoring Time
// FB OPEN Time
      L     t#20s;
      T     #"AV-03.01".MON_T;
      T     #"AV-03.02".MON_T;
      T     #"AV-03.03".MON_T;
      T     #"AV-03.04".MON_T;
      T     #"AV-03.05".MON_T;
      T     #"AV-03.06".MON_T;
      T     #"AV-03.07".MON_T;
      T     #"AV-03.08".MON_T;
      T     #"AV-03.09".MON_T;
      T     #"AV-03.10".MON_T;
      T     #"AV-03.11".MON_T;
      T     #"AV-03.12".MON_T;
      T     #"AV-03.13".MON_T;
      T     #"AV-03.14".MON_T;
      T     #"AV-03.15".MON_T;
// FB CLOSE Time
      L     t#20s;
      T     #"AV-03.01".MON_T_CLOSE;
      T     #"AV-03.02".MON_T_CLOSE;
      T     #"AV-03.03".MON_T_CLOSE;
      T     #"AV-03.04".MON_T_CLOSE;
      T     #"AV-03.05".MON_T_CLOSE;
      T     #"AV-03.06".MON_T_CLOSE;
      T     #"AV-03.07".MON_T_CLOSE;
      T     #"AV-03.08".MON_T_CLOSE;
      T     #"AV-03.09".MON_T_CLOSE;
      T     #"AV-03.10".MON_T_CLOSE;
      T     #"AV-03.11".MON_T_CLOSE;
      T     #"AV-03.12".MON_T_CLOSE;
      T     #"AV-03.13".MON_T_CLOSE;
      T     #"AV-03.14".MON_T_CLOSE;
      T     #"AV-03.15".MON_T_CLOSE;

REGION Network 3: AV-03.01 w ZSC
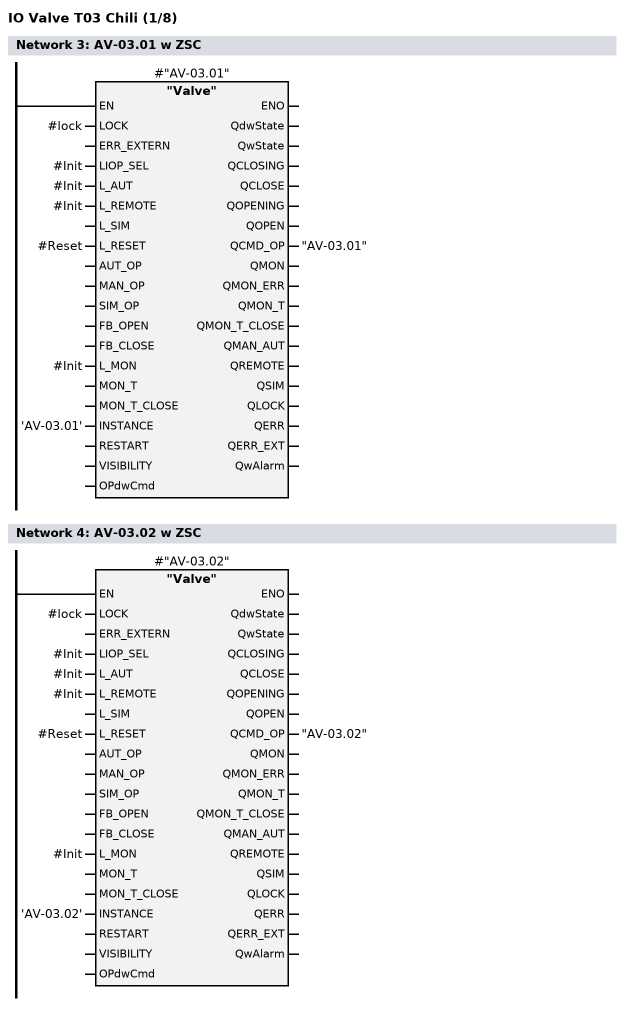
   RUNG wire#powerrail
      #"AV-03.01"(LOCK := #lock, ERR_EXTERN :=, LIOP_SEL := #Init, L_AUT := #Init, L_REMOTE := #Init, L_SIM :=, L_RESET := #Reset, AUT_OP :=, MAN_OP :=, SIM_OP :=, FB_OPEN :=, FB_CLOSE :=, L_MON := #Init, MON_T :=, MON_T_CLOSE :=, INSTANCE := 'AV-03.01', RESTART :=, VISIBILITY :=, OPdwCmd :=, QdwState =>, QwState =>, QCLOSING =>, QCLOSE =>, QOPENING =>, QOPEN =>, QCMD_OP => "AV-03.01", QMON =>, QMON_ERR =>, QMON_T =>, QMON_T_CLOSE =>, QMAN_AUT =>, QREMOTE =>, QSIM =>, QLOCK =>, QERR =>, QERR_EXT =>, QwAlarm =>)
   END_RUNG
   // the same network as SCL:
   #"AV-03.01"(LOCK := #lock,   // "Valve"
               LIOP_SEL := #Init,
               L_AUT := #Init,
               L_REMOTE := #Init,
               L_RESET := #Reset,
               L_MON := #Init,
               INSTANCE := 'AV-03.01',
               QCMD_OP => "AV-03.01");
END_REGION

REGION Network 4: AV-03.02 w ZSC
   RUNG wire#powerrail
      #"AV-03.02"(LOCK := #lock, ERR_EXTERN :=, LIOP_SEL := #Init, L_AUT := #Init, L_REMOTE := #Init, L_SIM :=, L_RESET := #Reset, AUT_OP :=, MAN_OP :=, SIM_OP :=, FB_OPEN :=, FB_CLOSE :=, L_MON := #Init, MON_T :=, MON_T_CLOSE :=, INSTANCE := 'AV-03.02', RESTART :=, VISIBILITY :=, OPdwCmd :=, QdwState =>, QwState =>, QCLOSING =>, QCLOSE =>, QOPENING =>, QOPEN =>, QCMD_OP => "AV-03.02", QMON =>, QMON_ERR =>, QMON_T =>, QMON_T_CLOSE =>, QMAN_AUT =>, QREMOTE =>, QSIM =>, QLOCK =>, QERR =>, QERR_EXT =>, QwAlarm =>)
   END_RUNG
   // the same network as SCL:
   #"AV-03.02"(LOCK := #lock,   // "Valve"
               LIOP_SEL := #Init,
               L_AUT := #Init,
               L_REMOTE := #Init,
               L_RESET := #Reset,
               L_MON := #Init,
               INSTANCE := 'AV-03.02',
               QCMD_OP => "AV-03.02");
END_REGION

REGION Network 5: AV-03.03 w ZSC
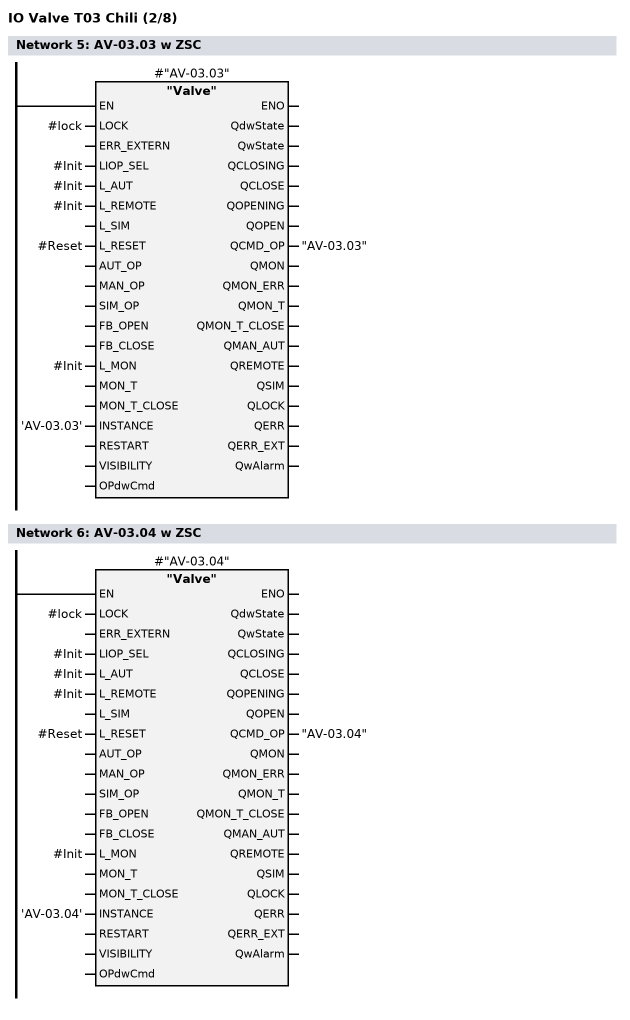
   RUNG wire#powerrail
      #"AV-03.03"(LOCK := #lock, ERR_EXTERN :=, LIOP_SEL := #Init, L_AUT := #Init, L_REMOTE := #Init, L_SIM :=, L_RESET := #Reset, AUT_OP :=, MAN_OP :=, SIM_OP :=, FB_OPEN :=, FB_CLOSE :=, L_MON := #Init, MON_T :=, MON_T_CLOSE :=, INSTANCE := 'AV-03.03', RESTART :=, VISIBILITY :=, OPdwCmd :=, QdwState =>, QwState =>, QCLOSING =>, QCLOSE =>, QOPENING =>, QOPEN =>, QCMD_OP => "AV-03.03", QMON =>, QMON_ERR =>, QMON_T =>, QMON_T_CLOSE =>, QMAN_AUT =>, QREMOTE =>, QSIM =>, QLOCK =>, QERR =>, QERR_EXT =>, QwAlarm =>)
   END_RUNG
   // the same network as SCL:
   #"AV-03.03"(LOCK := #lock,   // "Valve"
               LIOP_SEL := #Init,
               L_AUT := #Init,
               L_REMOTE := #Init,
               L_RESET := #Reset,
               L_MON := #Init,
               INSTANCE := 'AV-03.03',
               QCMD_OP => "AV-03.03");
END_REGION

REGION Network 6: AV-03.04 w ZSC
   RUNG wire#powerrail
      #"AV-03.04"(LOCK := #lock, ERR_EXTERN :=, LIOP_SEL := #Init, L_AUT := #Init, L_REMOTE := #Init, L_SIM :=, L_RESET := #Reset, AUT_OP :=, MAN_OP :=, SIM_OP :=, FB_OPEN :=, FB_CLOSE :=, L_MON := #Init, MON_T :=, MON_T_CLOSE :=, INSTANCE := 'AV-03.04', RESTART :=, VISIBILITY :=, OPdwCmd :=, QdwState =>, QwState =>, QCLOSING =>, QCLOSE =>, QOPENING =>, QOPEN =>, QCMD_OP => "AV-03.04", QMON =>, QMON_ERR =>, QMON_T =>, QMON_T_CLOSE =>, QMAN_AUT =>, QREMOTE =>, QSIM =>, QLOCK =>, QERR =>, QERR_EXT =>, QwAlarm =>)
   END_RUNG
   // the same network as SCL:
   #"AV-03.04"(LOCK := #lock,   // "Valve"
               LIOP_SEL := #Init,
               L_AUT := #Init,
               L_REMOTE := #Init,
               L_RESET := #Reset,
               L_MON := #Init,
               INSTANCE := 'AV-03.04',
               QCMD_OP => "AV-03.04");
END_REGION

REGION Network 7: AV-03.05
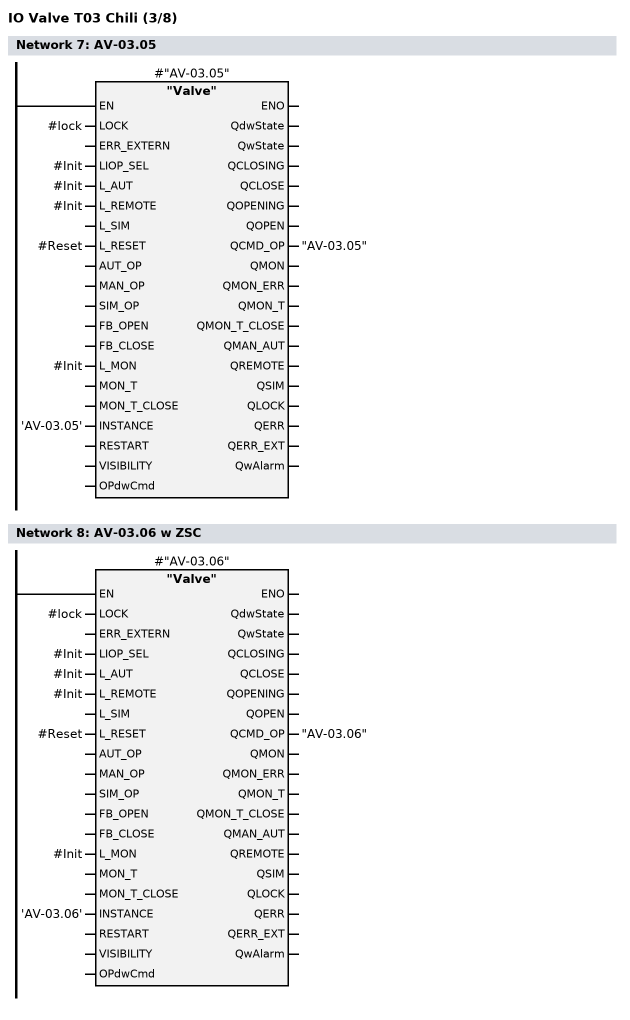
   RUNG wire#powerrail
      #"AV-03.05"(LOCK := #lock, ERR_EXTERN :=, LIOP_SEL := #Init, L_AUT := #Init, L_REMOTE := #Init, L_SIM :=, L_RESET := #Reset, AUT_OP :=, MAN_OP :=, SIM_OP :=, FB_OPEN :=, FB_CLOSE :=, L_MON := #Init, MON_T :=, MON_T_CLOSE :=, INSTANCE := 'AV-03.05', RESTART :=, VISIBILITY :=, OPdwCmd :=, QdwState =>, QwState =>, QCLOSING =>, QCLOSE =>, QOPENING =>, QOPEN =>, QCMD_OP => "AV-03.05", QMON =>, QMON_ERR =>, QMON_T =>, QMON_T_CLOSE =>, QMAN_AUT =>, QREMOTE =>, QSIM =>, QLOCK =>, QERR =>, QERR_EXT =>, QwAlarm =>)
   END_RUNG
   // the same network as SCL:
   #"AV-03.05"(LOCK := #lock,   // "Valve"
               LIOP_SEL := #Init,
               L_AUT := #Init,
               L_REMOTE := #Init,
               L_RESET := #Reset,
               L_MON := #Init,
               INSTANCE := 'AV-03.05',
               QCMD_OP => "AV-03.05");
END_REGION

REGION Network 8: AV-03.06 w ZSC
   RUNG wire#powerrail
      #"AV-03.06"(LOCK := #lock, ERR_EXTERN :=, LIOP_SEL := #Init, L_AUT := #Init, L_REMOTE := #Init, L_SIM :=, L_RESET := #Reset, AUT_OP :=, MAN_OP :=, SIM_OP :=, FB_OPEN :=, FB_CLOSE :=, L_MON := #Init, MON_T :=, MON_T_CLOSE :=, INSTANCE := 'AV-03.06', RESTART :=, VISIBILITY :=, OPdwCmd :=, QdwState =>, QwState =>, QCLOSING =>, QCLOSE =>, QOPENING =>, QOPEN =>, QCMD_OP => "AV-03.06", QMON =>, QMON_ERR =>, QMON_T =>, QMON_T_CLOSE =>, QMAN_AUT =>, QREMOTE =>, QSIM =>, QLOCK =>, QERR =>, QERR_EXT =>, QwAlarm =>)
   END_RUNG
   // the same network as SCL:
   #"AV-03.06"(LOCK := #lock,   // "Valve"
               LIOP_SEL := #Init,
               L_AUT := #Init,
               L_REMOTE := #Init,
               L_RESET := #Reset,
               L_MON := #Init,
               INSTANCE := 'AV-03.06',
               QCMD_OP => "AV-03.06");
END_REGION

REGION Network 9: AV-03.07
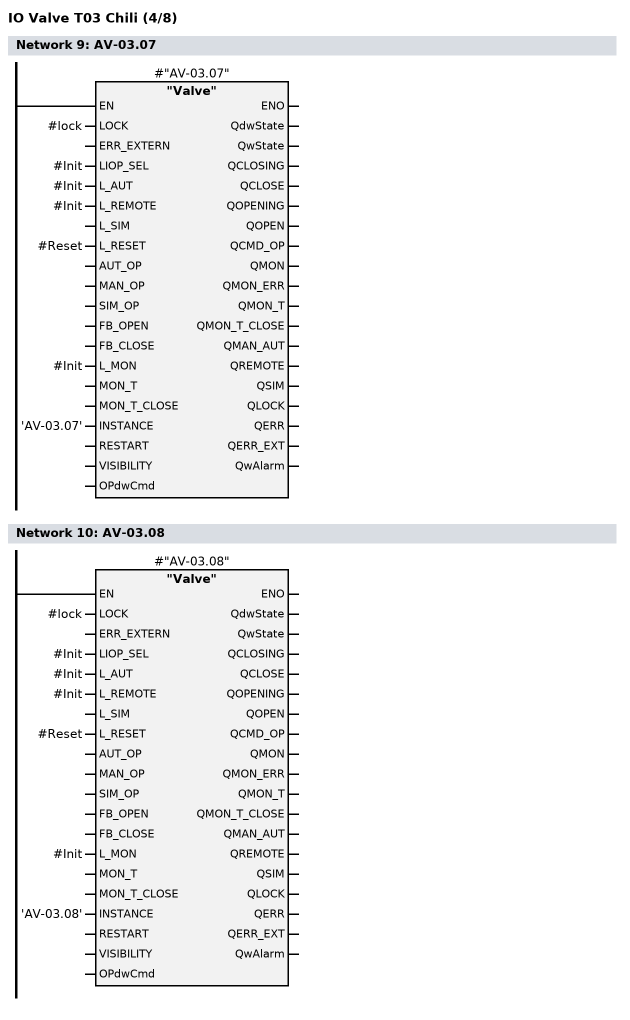
   RUNG wire#powerrail
      #"AV-03.07"(LOCK := #lock, ERR_EXTERN :=, LIOP_SEL := #Init, L_AUT := #Init, L_REMOTE := #Init, L_SIM :=, L_RESET := #Reset, AUT_OP :=, MAN_OP :=, SIM_OP :=, FB_OPEN :=, FB_CLOSE :=, L_MON := #Init, MON_T :=, MON_T_CLOSE :=, INSTANCE := 'AV-03.07', RESTART :=, VISIBILITY :=, OPdwCmd :=, QdwState =>, QwState =>, QCLOSING =>, QCLOSE =>, QOPENING =>, QOPEN =>, QCMD_OP =>, QMON =>, QMON_ERR =>, QMON_T =>, QMON_T_CLOSE =>, QMAN_AUT =>, QREMOTE =>, QSIM =>, QLOCK =>, QERR =>, QERR_EXT =>, QwAlarm =>)
   END_RUNG
   // the same network as SCL:
   #"AV-03.07"(LOCK := #lock,   // "Valve"
               LIOP_SEL := #Init,
               L_AUT := #Init,
               L_REMOTE := #Init,
               L_RESET := #Reset,
               L_MON := #Init,
               INSTANCE := 'AV-03.07');
END_REGION

REGION Network 10: AV-03.08
   RUNG wire#powerrail
      #"AV-03.08"(LOCK := #lock, ERR_EXTERN :=, LIOP_SEL := #Init, L_AUT := #Init, L_REMOTE := #Init, L_SIM :=, L_RESET := #Reset, AUT_OP :=, MAN_OP :=, SIM_OP :=, FB_OPEN :=, FB_CLOSE :=, L_MON := #Init, MON_T :=, MON_T_CLOSE :=, INSTANCE := 'AV-03.08', RESTART :=, VISIBILITY :=, OPdwCmd :=, QdwState =>, QwState =>, QCLOSING =>, QCLOSE =>, QOPENING =>, QOPEN =>, QCMD_OP =>, QMON =>, QMON_ERR =>, QMON_T =>, QMON_T_CLOSE =>, QMAN_AUT =>, QREMOTE =>, QSIM =>, QLOCK =>, QERR =>, QERR_EXT =>, QwAlarm =>)
   END_RUNG
   // the same network as SCL:
   #"AV-03.08"(LOCK := #lock,   // "Valve"
               LIOP_SEL := #Init,
               L_AUT := #Init,
               L_REMOTE := #Init,
               L_RESET := #Reset,
               L_MON := #Init,
               INSTANCE := 'AV-03.08');
END_REGION

REGION Network 11: AV-03.09
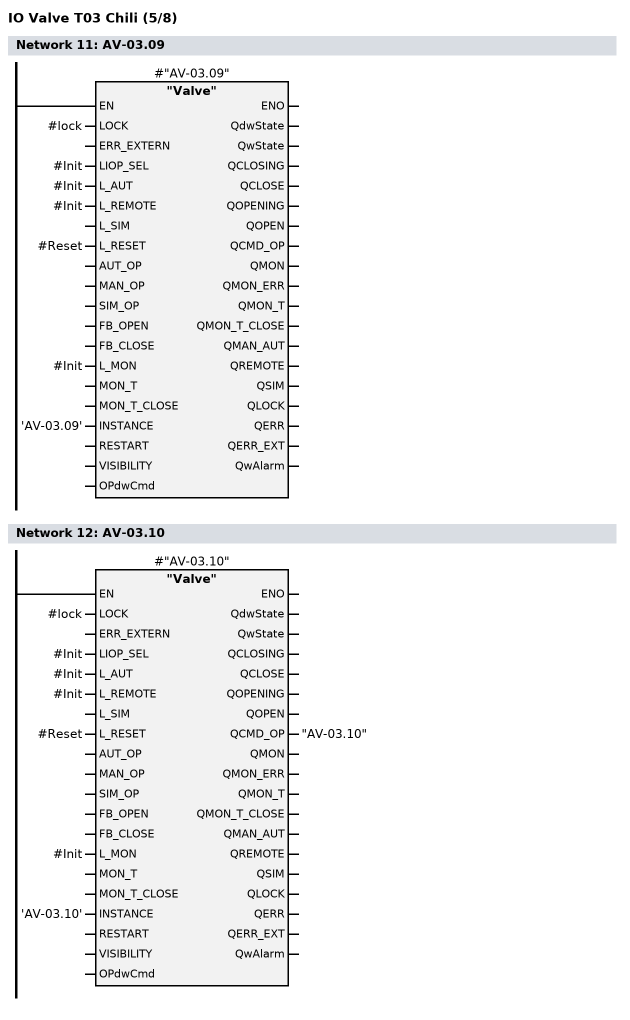
   RUNG wire#powerrail
      #"AV-03.09"(LOCK := #lock, ERR_EXTERN :=, LIOP_SEL := #Init, L_AUT := #Init, L_REMOTE := #Init, L_SIM :=, L_RESET := #Reset, AUT_OP :=, MAN_OP :=, SIM_OP :=, FB_OPEN :=, FB_CLOSE :=, L_MON := #Init, MON_T :=, MON_T_CLOSE :=, INSTANCE := 'AV-03.09', RESTART :=, VISIBILITY :=, OPdwCmd :=, QdwState =>, QwState =>, QCLOSING =>, QCLOSE =>, QOPENING =>, QOPEN =>, QCMD_OP =>, QMON =>, QMON_ERR =>, QMON_T =>, QMON_T_CLOSE =>, QMAN_AUT =>, QREMOTE =>, QSIM =>, QLOCK =>, QERR =>, QERR_EXT =>, QwAlarm =>)
   END_RUNG
   // the same network as SCL:
   #"AV-03.09"(LOCK := #lock,   // "Valve"
               LIOP_SEL := #Init,
               L_AUT := #Init,
               L_REMOTE := #Init,
               L_RESET := #Reset,
               L_MON := #Init,
               INSTANCE := 'AV-03.09');
END_REGION

REGION Network 12: AV-03.10
   RUNG wire#powerrail
      #"AV-03.10"(LOCK := #lock, ERR_EXTERN :=, LIOP_SEL := #Init, L_AUT := #Init, L_REMOTE := #Init, L_SIM :=, L_RESET := #Reset, AUT_OP :=, MAN_OP :=, SIM_OP :=, FB_OPEN :=, FB_CLOSE :=, L_MON := #Init, MON_T :=, MON_T_CLOSE :=, INSTANCE := 'AV-03.10', RESTART :=, VISIBILITY :=, OPdwCmd :=, QdwState =>, QwState =>, QCLOSING =>, QCLOSE =>, QOPENING =>, QOPEN =>, QCMD_OP => "AV-03.10", QMON =>, QMON_ERR =>, QMON_T =>, QMON_T_CLOSE =>, QMAN_AUT =>, QREMOTE =>, QSIM =>, QLOCK =>, QERR =>, QERR_EXT =>, QwAlarm =>)
   END_RUNG
   // the same network as SCL:
   #"AV-03.10"(LOCK := #lock,   // "Valve"
               LIOP_SEL := #Init,
               L_AUT := #Init,
               L_REMOTE := #Init,
               L_RESET := #Reset,
               L_MON := #Init,
               INSTANCE := 'AV-03.10',
               QCMD_OP => "AV-03.10");
END_REGION

REGION Network 13: AV-03.11 w ZSC
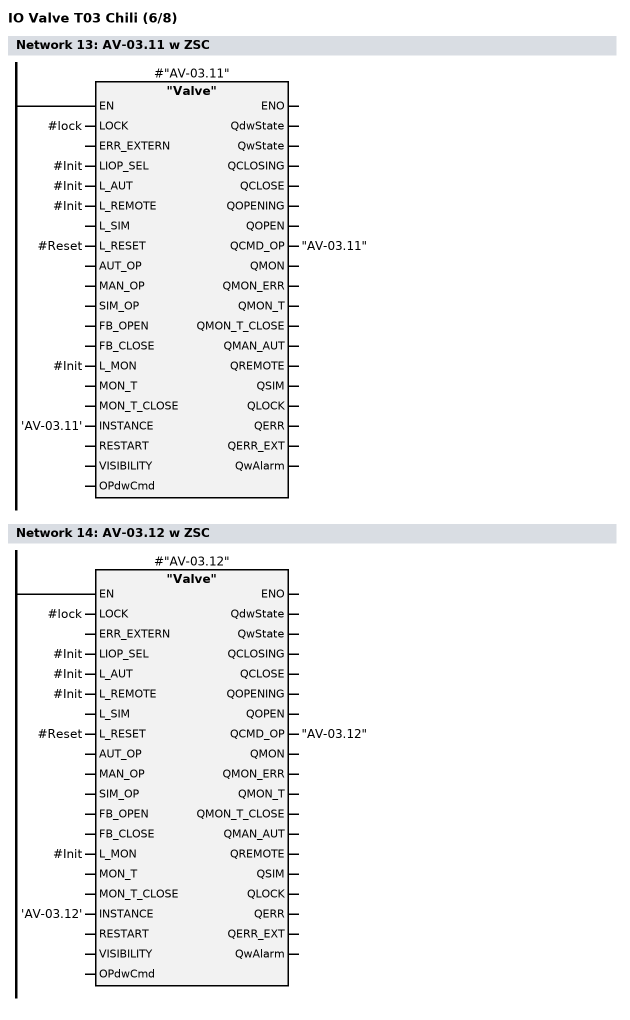
   RUNG wire#powerrail
      #"AV-03.11"(LOCK := #lock, ERR_EXTERN :=, LIOP_SEL := #Init, L_AUT := #Init, L_REMOTE := #Init, L_SIM :=, L_RESET := #Reset, AUT_OP :=, MAN_OP :=, SIM_OP :=, FB_OPEN :=, FB_CLOSE :=, L_MON := #Init, MON_T :=, MON_T_CLOSE :=, INSTANCE := 'AV-03.11', RESTART :=, VISIBILITY :=, OPdwCmd :=, QdwState =>, QwState =>, QCLOSING =>, QCLOSE =>, QOPENING =>, QOPEN =>, QCMD_OP => "AV-03.11", QMON =>, QMON_ERR =>, QMON_T =>, QMON_T_CLOSE =>, QMAN_AUT =>, QREMOTE =>, QSIM =>, QLOCK =>, QERR =>, QERR_EXT =>, QwAlarm =>)
   END_RUNG
   // the same network as SCL:
   #"AV-03.11"(LOCK := #lock,   // "Valve"
               LIOP_SEL := #Init,
               L_AUT := #Init,
               L_REMOTE := #Init,
               L_RESET := #Reset,
               L_MON := #Init,
               INSTANCE := 'AV-03.11',
               QCMD_OP => "AV-03.11");
END_REGION

REGION Network 14: AV-03.12 w ZSC
   RUNG wire#powerrail
      #"AV-03.12"(LOCK := #lock, ERR_EXTERN :=, LIOP_SEL := #Init, L_AUT := #Init, L_REMOTE := #Init, L_SIM :=, L_RESET := #Reset, AUT_OP :=, MAN_OP :=, SIM_OP :=, FB_OPEN :=, FB_CLOSE :=, L_MON := #Init, MON_T :=, MON_T_CLOSE :=, INSTANCE := 'AV-03.12', RESTART :=, VISIBILITY :=, OPdwCmd :=, QdwState =>, QwState =>, QCLOSING =>, QCLOSE =>, QOPENING =>, QOPEN =>, QCMD_OP => "AV-03.12", QMON =>, QMON_ERR =>, QMON_T =>, QMON_T_CLOSE =>, QMAN_AUT =>, QREMOTE =>, QSIM =>, QLOCK =>, QERR =>, QERR_EXT =>, QwAlarm =>)
   END_RUNG
   // the same network as SCL:
   #"AV-03.12"(LOCK := #lock,   // "Valve"
               LIOP_SEL := #Init,
               L_AUT := #Init,
               L_REMOTE := #Init,
               L_RESET := #Reset,
               L_MON := #Init,
               INSTANCE := 'AV-03.12',
               QCMD_OP => "AV-03.12");
END_REGION

REGION Network 15: AV-03.13 w ZSC
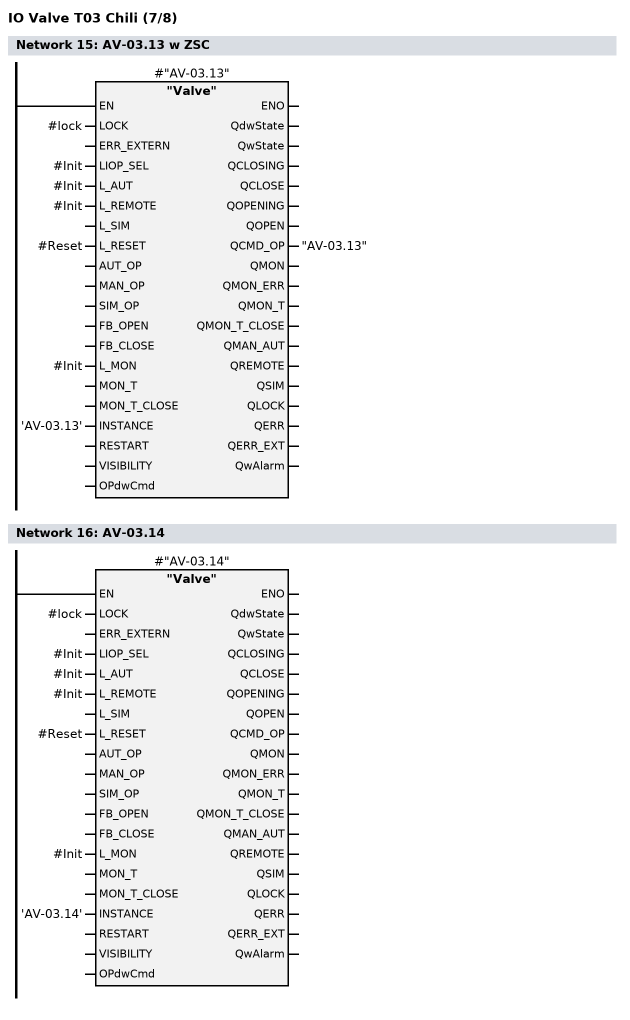
   RUNG wire#powerrail
      #"AV-03.13"(LOCK := #lock, ERR_EXTERN :=, LIOP_SEL := #Init, L_AUT := #Init, L_REMOTE := #Init, L_SIM :=, L_RESET := #Reset, AUT_OP :=, MAN_OP :=, SIM_OP :=, FB_OPEN :=, FB_CLOSE :=, L_MON := #Init, MON_T :=, MON_T_CLOSE :=, INSTANCE := 'AV-03.13', RESTART :=, VISIBILITY :=, OPdwCmd :=, QdwState =>, QwState =>, QCLOSING =>, QCLOSE =>, QOPENING =>, QOPEN =>, QCMD_OP => "AV-03.13", QMON =>, QMON_ERR =>, QMON_T =>, QMON_T_CLOSE =>, QMAN_AUT =>, QREMOTE =>, QSIM =>, QLOCK =>, QERR =>, QERR_EXT =>, QwAlarm =>)
   END_RUNG
   // the same network as SCL:
   #"AV-03.13"(LOCK := #lock,   // "Valve"
               LIOP_SEL := #Init,
               L_AUT := #Init,
               L_REMOTE := #Init,
               L_RESET := #Reset,
               L_MON := #Init,
               INSTANCE := 'AV-03.13',
               QCMD_OP => "AV-03.13");
END_REGION

REGION Network 16: AV-03.14
   RUNG wire#powerrail
      #"AV-03.14"(LOCK := #lock, ERR_EXTERN :=, LIOP_SEL := #Init, L_AUT := #Init, L_REMOTE := #Init, L_SIM :=, L_RESET := #Reset, AUT_OP :=, MAN_OP :=, SIM_OP :=, FB_OPEN :=, FB_CLOSE :=, L_MON := #Init, MON_T :=, MON_T_CLOSE :=, INSTANCE := 'AV-03.14', RESTART :=, VISIBILITY :=, OPdwCmd :=, QdwState =>, QwState =>, QCLOSING =>, QCLOSE =>, QOPENING =>, QOPEN =>, QCMD_OP =>, QMON =>, QMON_ERR =>, QMON_T =>, QMON_T_CLOSE =>, QMAN_AUT =>, QREMOTE =>, QSIM =>, QLOCK =>, QERR =>, QERR_EXT =>, QwAlarm =>)
   END_RUNG
   // the same network as SCL:
   #"AV-03.14"(LOCK := #lock,   // "Valve"
               LIOP_SEL := #Init,
               L_AUT := #Init,
               L_REMOTE := #Init,
               L_RESET := #Reset,
               L_MON := #Init,
               INSTANCE := 'AV-03.14');
END_REGION

REGION Network 17: AV-03.15
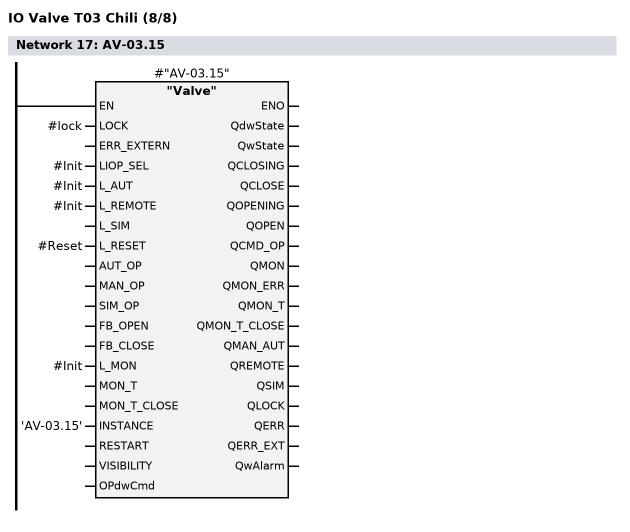
   RUNG wire#powerrail
      #"AV-03.15"(LOCK := #lock, ERR_EXTERN :=, LIOP_SEL := #Init, L_AUT := #Init, L_REMOTE := #Init, L_SIM :=, L_RESET := #Reset, AUT_OP :=, MAN_OP :=, SIM_OP :=, FB_OPEN :=, FB_CLOSE :=, L_MON := #Init, MON_T :=, MON_T_CLOSE :=, INSTANCE := 'AV-03.15', RESTART :=, VISIBILITY :=, OPdwCmd :=, QdwState =>, QwState =>, QCLOSING =>, QCLOSE =>, QOPENING =>, QOPEN =>, QCMD_OP =>, QMON =>, QMON_ERR =>, QMON_T =>, QMON_T_CLOSE =>, QMAN_AUT =>, QREMOTE =>, QSIM =>, QLOCK =>, QERR =>, QERR_EXT =>, QwAlarm =>)
   END_RUNG
   // the same network as SCL:
   #"AV-03.15"(LOCK := #lock,   // "Valve"
               LIOP_SEL := #Init,
               L_AUT := #Init,
               L_REMOTE := #Init,
               L_RESET := #Reset,
               L_MON := #Init,
               INSTANCE := 'AV-03.15');
END_REGION
END_FUNCTION_BLOCK

FUNCTION_BLOCK "IO Valve T04 Chili"   // FB304, LAD
{ S7_Optimized_Access := 'FALSE' }
VERSION : 0.1
// stored: AutoNumber false, IsIECCheckEnabled false, SetENOAutomatically false, UDAEnableTagReadback false
   VAR_INPUT
      lock : Bool;
      Init : Bool;
      testing : Bool;
      Reset : Bool;
   END_VAR
   VAR
      "AV-04.01" { S7_SetPoint := 'True'} : "Valve";   // AUTO BUTTERFLY VALVE INLET PROCESS WATER TO BFT CHILI AWETAN T-04.00
      "AV-04.02" { S7_SetPoint := 'True'} : "Valve";   // AUTO BUTTERFLY VALVE CIP SUPPLY TO BFT CHILI AWETAN T-04.00
      "AV-04.03" { S7_SetPoint := 'True'} : "Valve";   // AUTO BUTTERFLY VALVE OUTLET PRODUCT FROM BFT CHILI AWETAN T-04.00
      "AV-04.04" { S7_SetPoint := 'True'} : "Valve";   // AUTO BUTTERFLY VALVE OUTLET CIP TANK & LINE CHILI AWETAN T-04.00
      "AV-04.05" { S7_SetPoint := 'True'} : "Valve";   // AUTO BUTTERFLY VALVE DRAIN MONO PUMP P-04.01
      "AV-04.06" { S7_SetPoint := 'True'} : "Valve";   // AUTO BUTTERFLY VALVE INLET PRODUCT TO BFT CHILI AWETAN T-04.00
      "AV-04.07" { S7_SetPoint := 'True'} : "Valve";   // AUTO BUTTERFLY VALVE INLET CHILI AWETAN FROM T-03.00 TO BLENDING TANK T-20.00
      "AV-04.08" { S7_SetPoint := 'True'} : "Valve";
      "AV-04.09" { S7_SetPoint := 'True'} : "Valve";
      "AV-04.10" { S7_SetPoint := 'True'} : "Valve";
      "AV-04.11" { S7_SetPoint := 'True'} : "Valve";
      "AV-04.12" { S7_SetPoint := 'True'} : "Valve";
      "AV-04.13" { S7_SetPoint := 'True'} : "Valve";
      "AV-04.14" { S7_SetPoint := 'True'} : "Valve";
      "AV-04.15" { S7_SetPoint := 'True'} : "Valve";
   END_VAR
BEGIN

REGION Network 1 (SCL): FB OPEN and CLOSE
   IF #testing THEN
       // Statement section IF
       #"AV-04.01".FB_OPEN := #"AV-04.01".QCMD_OP;
       #"AV-04.01".FB_CLOSE := NOT #"AV-04.01".QCMD_OP;
       #"AV-04.02".FB_OPEN := #"AV-04.02".QCMD_OP;
       #"AV-04.02".FB_CLOSE := NOT #"AV-04.02".QCMD_OP;
       #"AV-04.03".FB_OPEN := #"AV-04.03".QCMD_OP;
       #"AV-04.03".FB_CLOSE := NOT #"AV-04.03".QCMD_OP;
       #"AV-04.04".FB_OPEN := #"AV-04.04".QCMD_OP;
       #"AV-04.04".FB_CLOSE := NOT #"AV-04.04".QCMD_OP;
       #"AV-04.05".FB_OPEN := #"AV-04.05".QCMD_OP;
       #"AV-04.05".FB_CLOSE := NOT #"AV-04.05".QCMD_OP;
       #"AV-04.06".FB_OPEN := #"AV-04.06".QCMD_OP;
       #"AV-04.06".FB_CLOSE := NOT #"AV-04.06".QCMD_OP;
       #"AV-04.07".FB_OPEN := #"AV-04.07".QCMD_OP;
       #"AV-04.07".FB_CLOSE := NOT #"AV-04.07".QCMD_OP;
       #"AV-04.08".FB_OPEN := #"AV-04.08".QCMD_OP;
       #"AV-04.08".FB_CLOSE := NOT #"AV-04.08".QCMD_OP;
       #"AV-04.09".FB_OPEN := #"AV-04.09".QCMD_OP;
       #"AV-04.09".FB_CLOSE := NOT #"AV-04.09".QCMD_OP;
       #"AV-04.10".FB_OPEN := #"AV-04.10".QCMD_OP;
       #"AV-04.10".FB_CLOSE := NOT #"AV-04.10".QCMD_OP;
       #"AV-04.11".FB_OPEN := #"AV-04.11".QCMD_OP;
       #"AV-04.11".FB_CLOSE := NOT #"AV-04.11".QCMD_OP;
       #"AV-04.12".FB_OPEN := #"AV-04.12".QCMD_OP;
       #"AV-04.12".FB_CLOSE := NOT #"AV-04.12".QCMD_OP;
       #"AV-04.13".FB_OPEN := #"AV-04.13".QCMD_OP;
       #"AV-04.13".FB_CLOSE := NOT #"AV-04.13".QCMD_OP;
       #"AV-04.14".FB_OPEN := #"AV-04.14".QCMD_OP;
       #"AV-04.14".FB_CLOSE := NOT #"AV-04.14".QCMD_OP;
       #"AV-04.15".FB_OPEN := #"AV-04.15".QCMD_OP;
       #"AV-04.15".FB_CLOSE := NOT #"AV-04.15".QCMD_OP;
   ELSE
       // Statement section ELSE
       #"AV-04.01".FB_OPEN := NOT "ZSC-04.01";
       #"AV-04.01".FB_CLOSE := "ZSC-04.01";
       #"AV-04.02".FB_OPEN := NOT "ZSC-04.02";
       #"AV-04.02".FB_CLOSE := "ZSC-04.02";
       #"AV-04.03".FB_OPEN := NOT "ZSC-04.03";
       #"AV-04.03".FB_CLOSE := "ZSC-04.03";
       #"AV-04.04".FB_OPEN := NOT "ZSC-04.04";
       #"AV-04.04".FB_CLOSE := "ZSC-04.04";
       #"AV-04.05".FB_OPEN := #"AV-04.05".QCMD_OP;
       #"AV-04.05".FB_CLOSE := NOT #"AV-04.05".QCMD_OP;
       #"AV-04.06".FB_OPEN := NOT "ZSC-04.06";
       #"AV-04.06".FB_CLOSE := "ZSC-04.06";
       #"AV-04.07".FB_OPEN := #"AV-04.07".QCMD_OP;
       #"AV-04.07".FB_CLOSE := NOT #"AV-04.07".QCMD_OP;
       #"AV-04.08".FB_OPEN := #"AV-04.08".QCMD_OP;
       #"AV-04.08".FB_CLOSE := NOT #"AV-04.08".QCMD_OP;
       #"AV-04.09".FB_OPEN := #"AV-04.09".QCMD_OP;
       #"AV-04.09".FB_CLOSE := NOT #"AV-04.09".QCMD_OP;
       #"AV-04.10".FB_OPEN := #"AV-04.10".QCMD_OP;
       #"AV-04.10".FB_CLOSE := NOT #"AV-04.10".QCMD_OP;
       #"AV-04.11".FB_OPEN := NOT "ZSC-04.11";
       #"AV-04.11".FB_CLOSE := "ZSC-04.11";
       #"AV-04.12".FB_OPEN := NOT "ZSC-04.12";
       #"AV-04.12".FB_CLOSE := "ZSC-04.12";
       #"AV-04.13".FB_OPEN := NOT "ZSC-04.13";
       #"AV-04.13".FB_CLOSE := "ZSC-04.13";
       #"AV-04.14".FB_OPEN := #"AV-04.14".QCMD_OP;
       #"AV-04.14".FB_CLOSE := NOT #"AV-04.14".QCMD_OP;
       #"AV-04.15".FB_OPEN := #"AV-04.15".QCMD_OP;
       #"AV-04.15".FB_CLOSE := NOT #"AV-04.15".QCMD_OP;
   END_IF;
END_REGION

NETWORK
TITLE = FB Monitoring Time
// FB OPEN Time
      L     t#20s;
      T     #"AV-04.01".MON_T;
      T     #"AV-04.02".MON_T;
      T     #"AV-04.03".MON_T;
      T     #"AV-04.04".MON_T;
      T     #"AV-04.05".MON_T;
      T     #"AV-04.06".MON_T;
      T     #"AV-04.07".MON_T;
      T     #"AV-04.08".MON_T;
      T     #"AV-04.09".MON_T;
      T     #"AV-04.10".MON_T;
      T     #"AV-04.11".MON_T;
      T     #"AV-04.12".MON_T;
      T     #"AV-04.13".MON_T;
      T     #"AV-04.14".MON_T;
      T     #"AV-04.15".MON_T;
// FB CLOSE Time
      L     t#20s;
      T     #"AV-04.01".MON_T_CLOSE;
      T     #"AV-04.02".MON_T_CLOSE;
      T     #"AV-04.03".MON_T_CLOSE;
      T     #"AV-04.04".MON_T_CLOSE;
      T     #"AV-04.05".MON_T_CLOSE;
      T     #"AV-04.06".MON_T_CLOSE;
      T     #"AV-04.07".MON_T_CLOSE;
      T     #"AV-04.08".MON_T_CLOSE;
      T     #"AV-04.09".MON_T_CLOSE;
      T     #"AV-04.10".MON_T_CLOSE;
      T     #"AV-04.11".MON_T_CLOSE;
      T     #"AV-04.12".MON_T_CLOSE;
      T     #"AV-04.13".MON_T_CLOSE;
      T     #"AV-04.14".MON_T_CLOSE;
      T     #"AV-04.15".MON_T_CLOSE;

REGION Network 3: AV-04.01 w ZSC
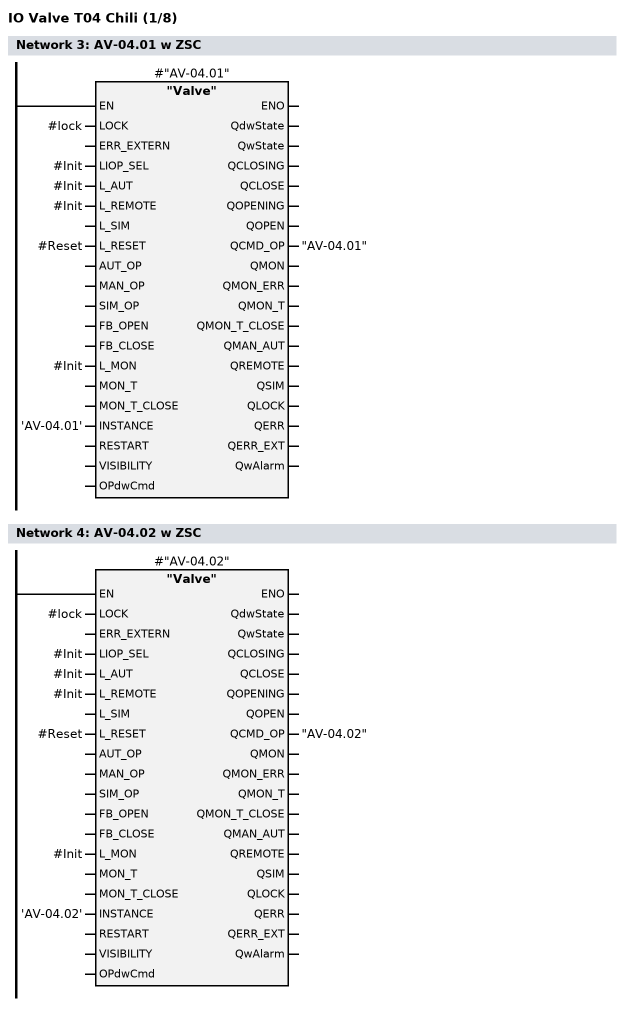
   RUNG wire#powerrail
      #"AV-04.01"(LOCK := #lock, ERR_EXTERN :=, LIOP_SEL := #Init, L_AUT := #Init, L_REMOTE := #Init, L_SIM :=, L_RESET := #Reset, AUT_OP :=, MAN_OP :=, SIM_OP :=, FB_OPEN :=, FB_CLOSE :=, L_MON := #Init, MON_T :=, MON_T_CLOSE :=, INSTANCE := 'AV-04.01', RESTART :=, VISIBILITY :=, OPdwCmd :=, QdwState =>, QwState =>, QCLOSING =>, QCLOSE =>, QOPENING =>, QOPEN =>, QCMD_OP => "AV-04.01", QMON =>, QMON_ERR =>, QMON_T =>, QMON_T_CLOSE =>, QMAN_AUT =>, QREMOTE =>, QSIM =>, QLOCK =>, QERR =>, QERR_EXT =>, QwAlarm =>)
   END_RUNG
   // the same network as SCL:
   #"AV-04.01"(LOCK := #lock,   // "Valve"
               LIOP_SEL := #Init,
               L_AUT := #Init,
               L_REMOTE := #Init,
               L_RESET := #Reset,
               L_MON := #Init,
               INSTANCE := 'AV-04.01',
               QCMD_OP => "AV-04.01");
END_REGION

REGION Network 4: AV-04.02 w ZSC
   RUNG wire#powerrail
      #"AV-04.02"(LOCK := #lock, ERR_EXTERN :=, LIOP_SEL := #Init, L_AUT := #Init, L_REMOTE := #Init, L_SIM :=, L_RESET := #Reset, AUT_OP :=, MAN_OP :=, SIM_OP :=, FB_OPEN :=, FB_CLOSE :=, L_MON := #Init, MON_T :=, MON_T_CLOSE :=, INSTANCE := 'AV-04.02', RESTART :=, VISIBILITY :=, OPdwCmd :=, QdwState =>, QwState =>, QCLOSING =>, QCLOSE =>, QOPENING =>, QOPEN =>, QCMD_OP => "AV-04.02", QMON =>, QMON_ERR =>, QMON_T =>, QMON_T_CLOSE =>, QMAN_AUT =>, QREMOTE =>, QSIM =>, QLOCK =>, QERR =>, QERR_EXT =>, QwAlarm =>)
   END_RUNG
   // the same network as SCL:
   #"AV-04.02"(LOCK := #lock,   // "Valve"
               LIOP_SEL := #Init,
               L_AUT := #Init,
               L_REMOTE := #Init,
               L_RESET := #Reset,
               L_MON := #Init,
               INSTANCE := 'AV-04.02',
               QCMD_OP => "AV-04.02");
END_REGION

REGION Network 5: AV-04.03 w ZSC
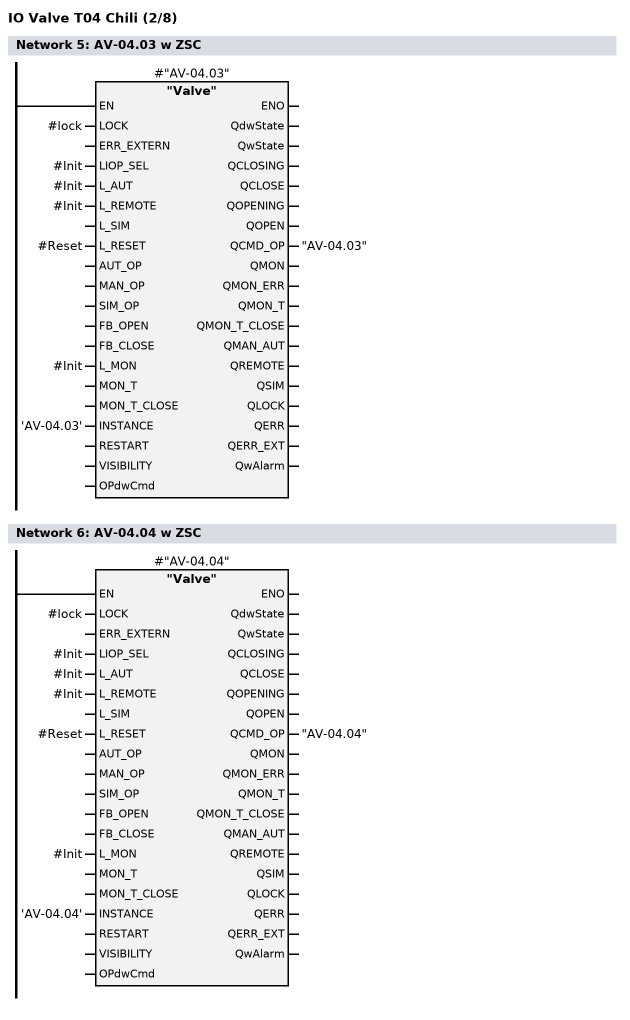
   RUNG wire#powerrail
      #"AV-04.03"(LOCK := #lock, ERR_EXTERN :=, LIOP_SEL := #Init, L_AUT := #Init, L_REMOTE := #Init, L_SIM :=, L_RESET := #Reset, AUT_OP :=, MAN_OP :=, SIM_OP :=, FB_OPEN :=, FB_CLOSE :=, L_MON := #Init, MON_T :=, MON_T_CLOSE :=, INSTANCE := 'AV-04.03', RESTART :=, VISIBILITY :=, OPdwCmd :=, QdwState =>, QwState =>, QCLOSING =>, QCLOSE =>, QOPENING =>, QOPEN =>, QCMD_OP => "AV-04.03", QMON =>, QMON_ERR =>, QMON_T =>, QMON_T_CLOSE =>, QMAN_AUT =>, QREMOTE =>, QSIM =>, QLOCK =>, QERR =>, QERR_EXT =>, QwAlarm =>)
   END_RUNG
   // the same network as SCL:
   #"AV-04.03"(LOCK := #lock,   // "Valve"
               LIOP_SEL := #Init,
               L_AUT := #Init,
               L_REMOTE := #Init,
               L_RESET := #Reset,
               L_MON := #Init,
               INSTANCE := 'AV-04.03',
               QCMD_OP => "AV-04.03");
END_REGION

REGION Network 6: AV-04.04 w ZSC
   RUNG wire#powerrail
      #"AV-04.04"(LOCK := #lock, ERR_EXTERN :=, LIOP_SEL := #Init, L_AUT := #Init, L_REMOTE := #Init, L_SIM :=, L_RESET := #Reset, AUT_OP :=, MAN_OP :=, SIM_OP :=, FB_OPEN :=, FB_CLOSE :=, L_MON := #Init, MON_T :=, MON_T_CLOSE :=, INSTANCE := 'AV-04.04', RESTART :=, VISIBILITY :=, OPdwCmd :=, QdwState =>, QwState =>, QCLOSING =>, QCLOSE =>, QOPENING =>, QOPEN =>, QCMD_OP => "AV-04.04", QMON =>, QMON_ERR =>, QMON_T =>, QMON_T_CLOSE =>, QMAN_AUT =>, QREMOTE =>, QSIM =>, QLOCK =>, QERR =>, QERR_EXT =>, QwAlarm =>)
   END_RUNG
   // the same network as SCL:
   #"AV-04.04"(LOCK := #lock,   // "Valve"
               LIOP_SEL := #Init,
               L_AUT := #Init,
               L_REMOTE := #Init,
               L_RESET := #Reset,
               L_MON := #Init,
               INSTANCE := 'AV-04.04',
               QCMD_OP => "AV-04.04");
END_REGION

REGION Network 7: AV-04.05
